LIN {X 0,Y 352.811,Z 516.095,A -85,B 0,C 180,E1 -17555.716,E2 -17555.716} C_VEL
LIN {X 0,Y 351.026,Z 514.823,A -85,B 0,C 180,E1 -17556.899,E2 -17556.899} C_VEL
LIN {X 0,Y 348.295,Z 512.255,A -85,B 0,C 180,E1 -17558.613,E2 -17558.613} C_VEL
LIN {X 0,Y 346.071,Z 510.125,A -85,B 0,C 180,E1 -17559.774,E2 -17559.774} C_VEL
LIN {X 0,Y 342.714,Z 507.631,A -85,B 0,C 180,E1 -17561.14,E2 -17561.14} C_VEL
LIN {X 0,Y 338.592,Z 503.953,A -85,B 0,C 180,E1 -17562.698,E2 -17562.698} C_VEL
LIN {X 0,Y 335.81,Z 501.368,A -85,B 0,C 180,E1 -17563.667,E2 -17563.667} C_VEL
LIN {X 0,Y 331.313,Z 497.271,A -85,B 0,C 180,E1 -17565.061,E2 -17565.061} C_VEL
LIN {X 0,Y 325.512,Z 491.626,A -85,B 0,C 180,E1 -17566.703,E2 -17566.703} C_VEL
LIN {X 0,Y 318.548,Z 484.573,A -85,B 0,C 180,E1 -17568.436,E2 -17568.436} C_VEL
LIN {X 0,Y 312.135,Z 477.632,A -85,B 0,C 180,E1 -17569.889,E2 -17569.889} C_VEL
LIN {X 0,Y 303.985,Z 468.251,A -85,B 0,C 180,E1 -17571.571,E2 -17571.571} C_VEL
LIN {X 0,Y 294.799,Z 456.635,A -85,B 0,C 180,E1 -17573.406,E2 -17573.406} C_VEL
LIN {X 0,Y 287.892,Z 445.985,A -85,B 0,C 180,E1 -17574.797,E2 -17574.797} C_VEL
LIN {X 0,Y 283.079,Z 436.29,A -85,B 0,C 180,E1 -17575.776,E2 -17575.776} C_VEL
LIN {X 0,Y 277.442,Z 424.043,A -85,B 0,C 180,E1 -17576.775,E2 -17576.775} C_VEL
LIN {X 0,Y 277.356,Z 423.437,A -85,B 0,C 180,E1 -17576.824,E2 -17576.824} C_VEL
LIN {X 0,Y 277.267,Z 423.447,A -85,B 0,C 180,E1 -17580.481,E2 -17580.481} C_VEL
LIN {X 0,Y 277.249,Z 423.45,A -85,B 0,C 180,E1 -17583.895,E2 -17583.895} C_VEL
LIN {X 0,Y 277.276,Z 423.448,A -85,B 0,C 180,E1 -17587.467,E2 -17587.467} C_VEL
LIN {X 0,Y 277.204,Z 423.456,A -85,B 0,C 180,E1 -17591.236,E2 -17591.236} C_VEL
LIN {X 0,Y 277.21,Z 423.456,A -85,B 0,C 180,E1 -17595.223,E2 -17595.223} C_VEL
LIN {X 0,Y 277.216,Z 423.454,A -85,B 0,C 180,E1 -17599.512,E2 -17599.512} C_VEL
LIN {X 0,Y 277.258,Z 423.447,A -85,B 0,C 180,E1 -17602.53,E2 -17602.53} C_VEL
LIN {X 0,Y 277.24,Z 423.448,A -85,B 0,C 180,E1 -17606.104,E2 -17606.104} C_VEL
LIN {X 0,Y 277.255,Z 423.448,A -85,B 0,C 180,E1 -17609.539,E2 -17609.539} C_VEL
LIN {X 0,Y 277.352,Z 423.439,A -85,B 0,C 180,E1 -17612.864,E2 -17612.864} C_VEL
LIN {X 0,Y 277.322,Z 423.437,A -85,B 0,C 180,E1 -17616.08,E2 -17616.08} C_VEL
LIN {X 0,Y 277.338,Z 423.436,A -85,B 0,C 180,E1 -17620.767,E2 -17620.767} C_VEL
LIN {X 0,Y 277.421,Z 423.424,A -85,B 0,C 180,E1 -17625.326,E2 -17625.326} C_VEL
LIN {X 0,Y 277.455,Z 423.42,A -85,B 0,C 180,E1 -17629.788,E2 -17629.788} C_VEL
LIN {X 0,Y 277.634,Z 423.404,A -85,B 0,C 180,E1 -17632.729,E2 -17632.729} C_VEL
LIN {X 0,Y 277.815,Z 423.365,A -85,B 0,C 180,E1 -17638.551,E2 -17638.551} C_VEL
LIN {X 0,Y 277.815,Z 423.375,A -85,B 0,C 180,E1 -17641.45,E2 -17641.45} C_VEL
LIN {X 0,Y 277.635,Z 423.4,A -85,B 0,C 180,E1 -17647.272,E2 -17647.272} C_VEL
LIN {X 0,Y 277.456,Z 423.426,A -85,B 0,C 180,E1 -17650.214,E2 -17650.214} C_VEL
LIN {X 0,Y 277.423,Z 423.429,A -85,B 0,C 180,E1 -17654.676,E2 -17654.676} C_VEL
LIN {X 0,Y 277.338,Z 423.437,A -85,B 0,C 180,E1 -17659.235,E2 -17659.235} C_VEL
LIN {X 0,Y 277.289,Z 423.449,A -85,B 0,C 180,E1 -17664.159,E2 -17664.159} C_VEL
LIN {X 0,Y 277.303,Z 423.44,A -85,B 0,C 180,E1 -17666.306,E2 -17666.306} C_VEL
LIN {X 0,Y 276.642,Z 423.527,A -85,B 0,C 180,E1 -17667.519,E2 -17667.519} C_VEL
LIN {X 0,Y 273.724,Z 423.89,A -85,B 0,C 180,E1 -17669.491,E2 -17669.491} C_VEL
LIN {X 0,Y 271.284,Z 424.343,A -85,B 0,C 180,E1 -17671.093,E2 -17671.093} C_VEL
LIN {X 0,Y 270.31,Z 424.816,A -85,B 0,C 180,E1 -17672.334,E2 -17672.334} C_VEL
LIN {X 0,Y 270.27,Z 425.007,A -85,B 0,C 180,E1 -17672.753,E2 -17672.753} C_VEL
LIN {X 0,Y 270.566,Z 427.131,A -85,B 0,C 180,E1 -17676.687,E2 -17676.687} C_VEL
LIN {X 0,Y 270.931,Z 429.384,A -85,B 0,C 180,E1 -17680.43,E2 -17680.43} C_VEL
LIN {X 0,Y 271.232,Z 432.01,A -85,B 0,C 180,E1 -17684.397,E2 -17684.397} C_VEL
LIN {X 0,Y 271.187,Z 434.37,A -85,B 0,C 180,E1 -17687.64,E2 -17687.64} C_VEL
LIN {X 0,Y 270.859,Z 437.105,A -85,B 0,C 180,E1 -17691.117,E2 -17691.117} C_VEL
LIN {X 0,Y 270.245,Z 440.416,A -85,B 0,C 180,E1 -17695.102,E2 -17695.102} C_VEL
LIN {X 0,Y 269.717,Z 443.488,A -85,B 0,C 180,E1 -17698.592,E2 -17698.592} C_VEL
LIN {X 0,Y 269.135,Z 447.13,A -85,B 0,C 180,E1 -17702.656,E2 -17702.656} C_VEL
LIN {X 0,Y 270.056,Z 450.505,A -85,B 0,C 180,E1 -17702.901,E2 -17702.901} C_VEL
LIN {X 0,Y 273.622,Z 464.1,A -85,B 0,C 180,E1 -17704.111,E2 -17704.111} C_VEL
LIN {X 0,Y 275.635,Z 473.958,A -85,B 0,C 180,E1 -17705.134,E2 -17705.134} C_VEL
LIN {X 0,Y 276.955,Z 484.089,A -85,B 0,C 180,E1 -17706.325,E2 -17706.325} C_VEL
LIN {X 0,Y 277.623,Z 492.133,A -85,B 0,C 180,E1 -17707.397,E2 -17707.397} C_VEL
LIN {X 0,Y 277.81,Z 496.843,A -85,B 0,C 180,E1 -17708.091,E2 -17708.091} C_VEL
LIN {X 0,Y 275.735,Z 508.341,A -85,B 0,C 180,E1 -17709.874,E2 -17709.874} C_VEL
LIN {X 0,Y 274.214,Z 516.042,A -85,B 0,C 180,E1 -17711.361,E2 -17711.361} C_VEL
LIN {X 0,Y 272.742,Z 523.682,A -85,B 0,C 180,E1 -17713.149,E2 -17713.149} C_VEL
LIN {X 0,Y 271.421,Z 530.22,A -85,B 0,C 180,E1 -17714.994,E2 -17714.994} C_VEL
LIN {X 0,Y 270.446,Z 534.72,A -85,B 0,C 180,E1 -17716.475,E2 -17716.475} C_VEL
LIN {X 0,Y 269.438,Z 540.214,A -85,B 0,C 180,E1 -17718.719,E2 -17718.719} C_VEL
LIN {X 0,Y 268.752,Z 544.542,A -85,B 0,C 180,E1 -17720.973,E2 -17720.973} C_VEL
LIN {X 0,Y 268.423,Z 546.911,A -85,B 0,C 180,E1 -17722.478,E2 -17722.478} C_VEL
LIN {X 0,Y 268.142,Z 549.611,A -85,B 0,C 180,E1 -17724.867,E2 -17724.867} C_VEL
LIN {X 0,Y 268.168,Z 551.166,A -85,B 0,C 180,E1 -17726.996,E2 -17726.996} C_VEL
LIN {X 0,Y 268.184,Z 551.757,A -85,B 0,C 180,E1 -17728.498,E2 -17728.498} C_VEL
LIN {X 0,Y 268.184,Z 551.757,A -85,B 0,C 180,E1 -17731.502,E2 -17731.502} C_VEL
LIN {X 0,Y 268.169,Z 551.166,A -85,B 0,C 180,E1 -17733.004,E2 -17733.004} C_VEL
LIN {X 0,Y 268.227,Z 548.712,A -85,B 0,C 180,E1 -17736.016,E2 -17736.016} C_VEL
LIN {X 0,Y 268.566,Z 545.76,A -85,B 0,C 180,E1 -17738.275,E2 -17738.275} C_VEL
LIN {X 0,Y 269.201,Z 541.77,A -85,B 0,C 180,E1 -17740.53,E2 -17740.53} C_VEL
LIN {X 0,Y 270.049,Z 536.636,A -85,B 0,C 180,E1 -17742.78,E2 -17742.78} C_VEL
LIN {X 0,Y 271.142,Z 531.374,A -85,B 0,C 180,E1 -17744.638,E2 -17744.638} C_VEL
LIN {X 0,Y 272.187,Z 526.434,A -85,B 0,C 180,E1 -17746.115,E2 -17746.115} C_VEL
LIN {X 0,Y 273.392,Z 520.735,A -85,B 0,C 180,E1 -17747.581,E2 -17747.581} C_VEL
LIN {X 0,Y 274.891,Z 512.177,A -85,B 0,C 180,E1 -17749.412,E2 -17749.412} C_VEL
LIN {X 0,Y 276.5,Z 504,A -85,B 0,C 180,E1 -17750.845,E2 -17750.845} C_VEL
LIN {X 0,Y 277.807,Z 496.842,A -85,B 0,C 180,E1 -17751.909,E2 -17751.909} C_VEL
LIN {X 0,Y 277.292,Z 487.688,A -85,B 0,C 180,E1 -17753.211,E2 -17753.211} C_VEL
LIN {X 0,Y 276.179,Z 477.496,A -85,B 0,C 180,E1 -17754.464,E2 -17754.464} C_VEL
LIN {X 0,Y 274.478,Z 467.955,A -85,B 0,C 180,E1 -17755.501,E2 -17755.501} C_VEL
LIN {X 0,Y 271.905,Z 457.255,A -85,B 0,C 180,E1 -17756.52,E2 -17756.52} C_VEL
LIN {X 0,Y 269.178,Z 447.606,A -85,B 0,C 180,E1 -17757.308,E2 -17757.308} C_VEL
LIN {X 0,Y 269.124,Z 447.099,A -85,B 0,C 180,E1 -17757.39,E2 -17757.39} C_VEL
LIN {X 0,Y 269.717,Z 443.392,A -85,B 0,C 180,E1 -17761.408,E2 -17761.408} C_VEL
LIN {X 0,Y 270.239,Z 440.375,A -85,B 0,C 180,E1 -17764.899,E2 -17764.899} C_VEL
LIN {X 0,Y 270.861,Z 437.075,A -85,B 0,C 180,E1 -17768.884,E2 -17768.884} C_VEL
LIN {X 0,Y 271.208,Z 434.364,A -85,B 0,C 180,E1 -17772.356,E2 -17772.356} C_VEL
LIN {X 0,Y 271.225,Z 432.001,A -85,B 0,C 180,E1 -17775.602,E2 -17775.602} C_VEL
LIN {X 0,Y 270.928,Z 429.377,A -85,B 0,C 180,E1 -17779.57,E2 -17779.57} C_VEL
LIN {X 0,Y 270.543,Z 426.938,A -85,B 0,C 180,E1 -17783.637,E2 -17783.637} C_VEL
LIN {X 0,Y 270.312,Z 425.167,A -85,B 0,C 180,E1 -17786.907,E2 -17786.907} C_VEL
LIN {X 0,Y 270.199,Z 424.332,A -85,B 0,C 180,E1 -17789.129,E2 -17789.129} C_VEL
LIN {X 0,Y 270.262,Z 424.322,A -85,B 0,C 180,E1 -17792.144,E2 -17792.144} C_VEL
LIN {X 0,Y 270.234,Z 424.325,A -85,B 0,C 180,E1 -17795.537,E2 -17795.537} C_VEL
LIN {X 0,Y 270.296,Z 424.316,A -85,B 0,C 180,E1 -17800.243,E2 -17800.243} C_VEL
LIN {X 0,Y 270.392,Z 424.302,A -85,B 0,C 180,E1 -17804.934,E2 -17804.934} C_VEL
LIN {X 0,Y 270.408,Z 424.304,A -85,B 0,C 180,E1 -17809.517,E2 -17809.517} C_VEL
LIN {X 0,Y 270.593,Z 424.276,A -85,B 0,C 180,E1 -17812.538,E2 -17812.538} C_VEL
LIN {X 0,Y 270.781,Z 424.251,A -85,B 0,C 180,E1 -17818.512,E2 -17818.512} C_VEL
LIN {X 0,Y 270.781,Z 424.239,A -85,B 0,C 180,E1 -17821.486,E2 -17821.486} C_VEL
LIN {X 0,Y 270.592,Z 424.28,A -85,B 0,C 180,E1 -17827.461,E2 -17827.461} C_VEL
LIN {X 0,Y 270.406,Z 424.298,A -85,B 0,C 180,E1 -17830.482,E2 -17830.482} C_VEL
LIN {X 0,Y 270.39,Z 424.301,A -85,B 0,C 180,E1 -17835.064,E2 -17835.064} C_VEL
LIN {X 0,Y 270.295,Z 424.311,A -85,B 0,C 180,E1 -17839.755,E2 -17839.755} C_VEL
LIN {X 0,Y 270.268,Z 424.317,A -85,B 0,C 180,E1 -17844.585,E2 -17844.585} C_VEL
LIN {X 0,Y 270.266,Z 424.317,A -85,B 0,C 180,E1 -17847.908,E2 -17847.908} C_VEL
LIN {X 0,Y 270.178,Z 424.33,A -85,B 0,C 180,E1 -17851.348,E2 -17851.348} C_VEL
LIN {X 0,Y 270.209,Z 424.328,A -85,B 0,C 180,E1 -17854.903,E2 -17854.903} C_VEL
LIN {X 0,Y 270.216,Z 424.326,A -85,B 0,C 180,E1 -17858.717,E2 -17858.717} C_VEL
LIN {X 0,Y 270.242,Z 424.324,A -85,B 0,C 180,E1 -17862.543,E2 -17862.543} C_VEL
LIN {X 0,Y 270.183,Z 424.331,A -85,B 0,C 180,E1 -17866.746,E2 -17866.746} C_VEL
LIN {X 0,Y 270.201,Z 424.327,A -85,B 0,C 180,E1 -17871.374,E2 -17871.374} C_VEL
LIN {X 0,Y 270.209,Z 424.327,A -85,B 0,C 180,E1 -17875.097,E2 -17875.097} C_VEL
LIN {X 0,Y 270.195,Z 424.328,A -85,B 0,C 180,E1 -17879.131,E2 -17879.131} C_VEL
LIN {X 0,Y 270.291,Z 424.318,A -85,B 0,C 180,E1 -17882.44,E2 -17882.44} C_VEL
LIN {X 0,Y 271.242,Z 427.063,A -85,B 0,C 180,E1 -17882.645,E2 -17882.645} C_VEL
LIN {X 0,Y 276.988,Z 439.088,A -85,B 0,C 180,E1 -17883.735,E2 -17883.735} C_VEL
LIN {X 0,Y 281.103,Z 447.875,A -85,B 0,C 180,E1 -17884.676,E2 -17884.676} C_VEL
LIN {X 0,Y 286.353,Z 456.735,A -85,B 0,C 180,E1 -17885.846,E2 -17885.846} C_VEL
LIN {X 0,Y 293.982,Z 467.207,A -85,B 0,C 180,E1 -17887.512,E2 -17887.512} C_VEL
LIN {X 0,Y 304.138,Z 479.227,A -85,B 0,C 180,E1 -17889.72,E2 -17889.72} C_VEL
LIN {X 0,Y 312.671,Z 488.513,A -85,B 0,C 180,E1 -17891.659,E2 -17891.659} C_VEL
LIN {X 0,Y 318.131,Z 494.088,A -85,B 0,C 180,E1 -17893.003,E2 -17893.003} C_VEL
LIN {X 0,Y 324.266,Z 500.008,A -85,B 0,C 180,E1 -17894.648,E2 -17894.648} C_VEL
LIN {X 0,Y 330.066,Z 505.438,A -85,B 0,C 180,E1 -17896.455,E2 -17896.455} C_VEL
LIN {X 0,Y 334.025,Z 509.236,A -85,B 0,C 180,E1 -17897.854,E2 -17897.854} C_VEL
LIN {X 0,Y 338.748,Z 513.032,A -85,B 0,C 180,E1 -17899.644,E2 -17899.644} C_VEL
LIN {X 0,Y 341.597,Z 515.35,A -85,B 0,C 180,E1 -17900.944,E2 -17900.944} C_VEL
LIN {X 0,Y 344.939,Z 518.614,A -85,B 0,C 180,E1 -17902.978,E2 -17902.978} C_VEL
LIN {X 0,Y 346.73,Z 519.995,A -85,B 0,C 180,E1 -17904.183,E2 -17904.183} C_VEL
LIN {X 0,Y 348.359,Z 520.945,A -85,B 0,C 180,E1 -17905.371,E2 -17905.371} C_VEL
LIN {X 0,Y 349.735,Z 521.553,A -85,B 0,C 180,E1 -17906.544,E2 -17906.544} C_VEL
LIN {X 0,Y 350.851,Z 521.883,A -85,B 0,C 180,E1 -17907.704,E2 -17907.704} C_VEL
LIN {X 0,Y 351.612,Z 522.025,A -85,B 0,C 180,E1 -17908.855,E2 -17908.855} C_VEL
LIN {X 0,Y 351.859,Z 522.078,A -85,B 0,C 180,E1 -17910,E2 -17910} C_VEL
LIN {X 0,Y 351.482,Z 522.043,A -85,B 0,C 180,E1 -17911.274,E2 -17911.274} C_VEL
LIN {X 0,Y 350.848,Z 521.881,A -85,B 0,C 180,E1 -17912.296,E2 -17912.296} C_VEL
LIN {X 0,Y 349.737,Z 521.547,A -85,B 0,C 180,E1 -17913.456,E2 -17913.456} C_VEL
LIN {X 0,Y 348.369,Z 520.948,A -85,B 0,C 180,E1 -17914.628,E2 -17914.628} C_VEL
LIN {X 0,Y 346.329,Z 519.696,A -85,B 0,C 180,E1 -17916.101,E2 -17916.101} C_VEL
LIN {X 0,Y 342.974,Z 516.792,A -85,B 0,C 180,E1 -17918.247,E2 -17918.247} C_VEL
LIN {X 0,Y 340.695,Z 514.539,A -85,B 0,C 180,E1 -17919.499,E2 -17919.499} C_VEL
LIN {X 0,Y 336.656,Z 511.495,A -85,B 0,C 180,E1 -17921.141,E2 -17921.141} C_VEL
LIN {X 0,Y 333.351,Z 508.557,A -85,B 0,C 180,E1 -17922.398,E2 -17922.398} C_VEL
LIN {X 0,Y 328.67,Z 504.29,A -85,B 0,C 180,E1 -17923.98,E2 -17923.98} C_VEL
LIN {X 0,Y 323.217,Z 499.024,A -85,B 0,C 180,E1 -17925.645,E2 -17925.645} C_VEL
LIN {X 0,Y 316.655,Z 492.581,A -85,B 0,C 180,E1 -17927.379,E2 -17927.379} C_VEL
LIN {X 0,Y 309.448,Z 484.978,A -85,B 0,C 180,E1 -17929.097,E2 -17929.097} C_VEL
LIN {X 0,Y 301.038,Z 475.669,A -85,B 0,C 180,E1 -17930.962,E2 -17930.962} C_VEL
LIN {X 0,Y 291.455,Z 463.927,A -85,B 0,C 180,E1 -17933.036,E2 -17933.036} C_VEL
LIN {X 0,Y 284.677,Z 454.079,A -85,B 0,C 180,E1 -17934.522,E2 -17934.522} C_VEL
LIN {X 0,Y 279.845,Z 445.412,A -85,B 0,C 180,E1 -17935.614,E2 -17935.614} C_VEL
LIN {X 0,Y 273.844,Z 432.334,A -85,B 0,C 180,E1 -17936.893,E2 -17936.893} C_VEL
LIN {X 0,Y 270.474,Z 425.245,A -85,B 0,C 180,E1 -17937.493,E2 -17937.493} C_VEL
LIN {X 0,Y 270.278,Z 424.32,A -85,B 0,C 180,E1 -17937.59,E2 -17937.59} C_VEL
LIN {X 0,Y 270.179,Z 424.332,A -85,B 0,C 180,E1 -17941.348,E2 -17941.348} C_VEL
LIN {X 0,Y 270.209,Z 424.327,A -85,B 0,C 180,E1 -17944.903,E2 -17944.903} C_VEL
LIN {X 0,Y 270.217,Z 424.325,A -85,B 0,C 180,E1 -17948.717,E2 -17948.717} C_VEL
LIN {X 0,Y 270.166,Z 424.333,A -85,B 0,C 180,E1 -17953.25,E2 -17953.25} C_VEL
LIN {X 0,Y 270.168,Z 424.333,A -85,B 0,C 180,E1 -17957.442,E2 -17957.442} C_VEL
LIN {X 0,Y 270.201,Z 424.328,A -85,B 0,C 180,E1 -17961.374,E2 -17961.374} C_VEL
LIN {X 0,Y 270.195,Z 424.33,A -85,B 0,C 180,E1 -17965.095,E2 -17965.095} C_VEL
LIN {X 0,Y 270.194,Z 424.33,A -85,B 0,C 180,E1 -17969.131,E2 -17969.131} C_VEL
LIN {X 0,Y 270.259,Z 424.318,A -85,B 0,C 180,E1 -17972.146,E2 -17972.146} C_VEL
LIN {X 0,Y 270.271,Z 424.316,A -85,B 0,C 180,E1 -17975.52,E2 -17975.52} C_VEL
LIN {X 0,Y 270.295,Z 424.311,A -85,B 0,C 180,E1 -17980.245,E2 -17980.245} C_VEL
LIN {X 0,Y 270.39,Z 424.301,A -85,B 0,C 180,E1 -17984.936,E2 -17984.936} C_VEL
LIN {X 0,Y 270.406,Z 424.298,A -85,B 0,C 180,E1 -17989.518,E2 -17989.518} C_VEL
LIN {X 0,Y 270.592,Z 424.28,A -85,B 0,C 180,E1 -17992.539,E2 -17992.539} C_VEL
LIN {X 0,Y 270.781,Z 424.239,A -85,B 0,C 180,E1 -17998.514,E2 -17998.514} C_VEL
LIN {X 0,Y 270.781,Z 424.251,A -85,B 0,C 180,E1 -18001.488,E2 -18001.488} C_VEL
LIN {X 0,Y 270.593,Z 424.277,A -85,B 0,C 180,E1 -18007.462,E2 -18007.462} C_VEL
LIN {X 0,Y 270.408,Z 424.304,A -85,B 0,C 180,E1 -18010.483,E2 -18010.483} C_VEL
LIN {X 0,Y 270.392,Z 424.303,A -85,B 0,C 180,E1 -18015.066,E2 -18015.066} C_VEL
LIN {X 0,Y 270.296,Z 424.316,A -85,B 0,C 180,E1 -18019.757,E2 -18019.757} C_VEL
LIN {X 0,Y 270.235,Z 424.325,A -85,B 0,C 180,E1 -18024.59,E2 -18024.59} C_VEL
LIN {X 0,Y 270.269,Z 424.321,A -85,B 0,C 180,E1 -18027.91,E2 -18027.91} C_VEL
LIN {X 0,Y 270.188,Z 424.334,A -85,B 0,C 180,E1 -18031.349,E2 -18031.349} C_VEL
LIN {X 0,Y 270.27,Z 425.007,A -85,B 0,C 180,E1 -18032.753,E2 -18032.753} C_VEL
LIN {X 0,Y 269.725,Z 425.745,A -85,B 0,C 180,E1 -18033.99,E2 -18033.99} C_VEL
LIN {X 0,Y 267,Z 427.276,A -85,B 0,C 180,E1 -18036,E2 -18036} C_VEL
LIN {X 0,Y 264.697,Z 428.566,A -85,B 0,C 180,E1 -18037.633,E2 -18037.633} C_VEL
LIN {X 0,Y 263.806,Z 429.451,A -85,B 0,C 180,E1 -18038.899,E2 -18038.899} C_VEL
LIN {X 0,Y 263.789,Z 429.714,A -85,B 0,C 180,E1 -18039.327,E2 -18039.327} C_VEL
LIN {X 0,Y 264.01,Z 431.244,A -85,B 0,C 180,E1 -18041.811,E2 -18041.811} C_VEL
LIN {X 0,Y 264.165,Z 432.745,A -85,B 0,C 180,E1 -18044.085,E2 -18044.085} C_VEL
LIN {X 0,Y 264.192,Z 434.229,A -85,B 0,C 180,E1 -18046.24,E2 -18046.24} C_VEL
LIN {X 0,Y 264.113,Z 435.726,A -85,B 0,C 180,E1 -18048.3,E2 -18048.3} C_VEL
LIN {X 0,Y 263.871,Z 437.477,A -85,B 0,C 180,E1 -18050.57,E2 -18050.57} C_VEL
LIN {X 0,Y 263.321,Z 440.252,A -85,B 0,C 180,E1 -18054.044,E2 -18054.044} C_VEL
LIN {X 0,Y 262.778,Z 443.322,A -85,B 0,C 180,E1 -18057.664,E2 -18057.664} C_VEL
LIN {X 0,Y 262.166,Z 446.678,A -85,B 0,C 180,E1 -18061.563,E2 -18061.563} C_VEL
LIN {X 0,Y 262.146,Z 446.972,A -85,B 0,C 180,E1 -18061.878,E2 -18061.878} C_VEL
LIN {X 0,Y 262.916,Z 450.048,A -85,B 0,C 180,E1 -18062.092,E2 -18062.092} C_VEL
LIN {X 0,Y 266.453,Z 462.719,A -85,B 0,C 180,E1 -18063.265,E2 -18063.265} C_VEL
LIN {X 0,Y 268.77,Z 473.748,A -85,B 0,C 180,E1 -18064.454,E2 -18064.454} C_VEL
LIN {X 0,Y 270.088,Z 483.277,A -85,B 0,C 180,E1 -18065.61,E2 -18065.61} C_VEL
LIN {X 0,Y 270.825,Z 492.155,A -85,B 0,C 180,E1 -18066.831,E2 -18066.831} C_VEL
LIN {X 0,Y 271.007,Z 497.997,A -85,B 0,C 180,E1 -18067.712,E2 -18067.712} C_VEL
LIN {X 0,Y 269.064,Z 508.143,A -85,B 0,C 180,E1 -18069.353,E2 -18069.353} C_VEL
LIN {X 0,Y 267.261,Z 516.833,A -85,B 0,C 180,E1 -18071.099,E2 -18071.099} C_VEL
LIN {X 0,Y 265.949,Z 523.484,A -85,B 0,C 180,E1 -18072.705,E2 -18072.705} C_VEL
LIN {X 0,Y 264.543,Z 530.022,A -85,B 0,C 180,E1 -18074.594,E2 -18074.594} C_VEL
LIN {X 0,Y 263.533,Z 534.522,A -85,B 0,C 180,E1 -18076.113,E2 -18076.113} C_VEL
LIN {X 0,Y 262.443,Z 540.016,A -85,B 0,C 180,E1 -18078.414,E2 -18078.414} C_VEL
LIN {X 0,Y 261.726,Z 544.345,A -85,B 0,C 180,E1 -18080.729,E2 -18080.729} C_VEL
LIN {X 0,Y 261.359,Z 546.713,A -85,B 0,C 180,E1 -18082.273,E2 -18082.273} C_VEL
LIN {X 0,Y 261.043,Z 549.602,A -85,B 0,C 180,E1 -18084.973,E2 -18084.973} C_VEL
LIN {X 0,Y 261.063,Z 550.968,A -85,B 0,C 180,E1 -18086.914,E2 -18086.914} C_VEL
LIN {X 0,Y 261.09,Z 551.56,A -85,B 0,C 180,E1 -18088.458,E2 -18088.458} C_VEL
LIN {X 0,Y 261.127,Z 551.716,A -85,B 0,C 180,E1 -18090,E2 -18090} C_VEL
LIN {X 0,Y 261.09,Z 551.56,A -85,B 0,C 180,E1 -18091.542,E2 -18091.542} C_VEL
LIN {X 0,Y 261.064,Z 550.968,A -85,B 0,C 180,E1 -18093.086,E2 -18093.086} C_VEL
LIN {X 0,Y 261.154,Z 548.515,A -85,B 0,C 180,E1 -18096.179,E2 -18096.179} C_VEL
LIN {X 0,Y 261.53,Z 545.563,A -85,B 0,C 180,E1 -18098.499,E2 -18098.499} C_VEL
LIN {X 0,Y 262.174,Z 541.571,A -85,B 0,C 180,E1 -18100.815,E2 -18100.815} C_VEL
LIN {X 0,Y 263.107,Z 536.438,A -85,B 0,C 180,E1 -18103.123,E2 -18103.123} C_VEL
LIN {X 0,Y 264.262,Z 531.177,A -85,B 0,C 180,E1 -18105.028,E2 -18105.028} C_VEL
LIN {X 0,Y 265.607,Z 524.859,A -85,B 0,C 180,E1 -18106.921,E2 -18106.921} C_VEL
LIN {X 0,Y 266.865,Z 518.908,A -85,B 0,C 180,E1 -18108.422,E2 -18108.422} C_VEL
LIN {X 0,Y 268.178,Z 511.979,A -85,B 0,C 180,E1 -18109.918,E2 -18109.918} C_VEL
LIN {X 0,Y 269.852,Z 503.802,A -85,B 0,C 180,E1 -18111.383,E2 -18111.383} C_VEL
LIN {X 0,Y 270.994,Z 497.997,A -85,B 0,C 180,E1 -18112.289,E2 -18112.289} C_VEL
LIN {X 0,Y 270.467,Z 487.254,A -85,B 0,C 180,E1 -18113.861,E2 -18113.861} C_VEL
LIN {X 0,Y 269.425,Z 477.778,A -85,B 0,C 180,E1 -18115.07,E2 -18115.07} C_VEL
LIN {X 0,Y 267.68,Z 468.336,A -85,B 0,C 180,E1 -18116.15,E2 -18116.15} C_VEL
LIN {X 0,Y 265.263,Z 458.078,A -85,B 0,C 180,E1 -18117.176,E2 -18117.176} C_VEL
LIN {X 0,Y 262.194,Z 447.497,A -85,B 0,C 180,E1 -18118.095,E2 -18118.095} C_VEL
LIN {X 0,Y 262.141,Z 446.947,A -85,B 0,C 180,E1 -18118.154,E2 -18118.154} C_VEL
LIN {X 0,Y 262.613,Z 444.306,A -85,B 0,C 180,E1 -18121.086,E2 -18121.086} C_VEL
LIN {X 0,Y 263.06,Z 441.747,A -85,B 0,C 180,E1 -18124.127,E2 -18124.127} C_VEL
LIN {X 0,Y 263.606,Z 438.712,A -85,B 0,C 180,E1 -18127.82,E2 -18127.82} C_VEL
LIN {X 0,Y 263.906,Z 437.223,A -85,B 0,C 180,E1 -18129.726,E2 -18129.726} C_VEL
LIN {X 0,Y 264.109,Z 435.628,A -85,B 0,C 180,E1 -18131.832,E2 -18131.832} C_VEL
LIN {X 0,Y 264.202,Z 433.988,A -85,B 0,C 180,E1 -18134.091,E2 -18134.091} C_VEL
LIN {X 0,Y 264.125,Z 432.517,A -85,B 0,C 180,E1 -18136.224,E2 -18136.224} C_VEL
LIN {X 0,Y 263.83,Z 429.957,A -85,B 0,C 180,E1 -18140.258,E2 -18140.258} C_VEL
LIN {X 0,Y 263.487,Z 427.756,A -85,B 0,C 180,E1 -18144.068,E2 -18144.068} C_VEL
LIN {X 0,Y 263.215,Z 425.859,A -85,B 0,C 180,E1 -18147.722,E2 -18147.722} C_VEL
LIN {X 0,Y 263.149,Z 425.21,A -85,B 0,C 180,E1 -18149.506,E2 -18149.506} C_VEL
LIN {X 0,Y 263.189,Z 425.201,A -85,B 0,C 180,E1 -18153.001,E2 -18153.001} C_VEL
LIN {X 0,Y 263.151,Z 425.207,A -85,B 0,C 180,E1 -18156.383,E2 -18156.383} C_VEL
LIN {X 0,Y 263.259,Z 425.195,A -85,B 0,C 180,E1 -18159.692,E2 -18159.692} C_VEL
LIN {X 0,Y 263.34,Z 425.181,A -85,B 0,C 180,E1 -18164.521,E2 -18164.521} C_VEL
LIN {X 0,Y 263.35,Z 425.181,A -85,B 0,C 180,E1 -18169.233,E2 -18169.233} C_VEL
LIN {X 0,Y 263.553,Z 425.153,A -85,B 0,C 180,E1 -18172.337,E2 -18172.337} C_VEL
LIN {X 0,Y 263.746,Z 425.127,A -85,B 0,C 180,E1 -18178.472,E2 -18178.472} C_VEL
LIN {X 0,Y 263.746,Z 425.114,A -85,B 0,C 180,E1 -18181.526,E2 -18181.526} C_VEL
LIN {X 0,Y 263.552,Z 425.155,A -85,B 0,C 180,E1 -18187.661,E2 -18187.661} C_VEL
LIN {X 0,Y 263.349,Z 425.178,A -85,B 0,C 180,E1 -18190.766,E2 -18190.766} C_VEL
LIN {X 0,Y 263.338,Z 425.181,A -85,B 0,C 180,E1 -18195.478,E2 -18195.478} C_VEL
LIN {X 0,Y 263.257,Z 425.187,A -85,B 0,C 180,E1 -18200.306,E2 -18200.306} C_VEL
LIN {X 0,Y 263.202,Z 425.197,A -85,B 0,C 180,E1 -18205.291,E2 -18205.291} C_VEL
LIN {X 0,Y 263.174,Z 425.203,A -85,B 0,C 180,E1 -18208.729,E2 -18208.729} C_VEL
LIN {X 0,Y 263.127,Z 425.208,A -85,B 0,C 180,E1 -18212.288,E2 -18212.288} C_VEL
LIN {X 0,Y 263.182,Z 425.199,A -85,B 0,C 180,E1 -18215.978,E2 -18215.978} C_VEL
LIN {X 0,Y 263.155,Z 425.203,A -85,B 0,C 180,E1 -18219.862,E2 -18219.862} C_VEL
LIN {X 0,Y 263.2,Z 425.198,A -85,B 0,C 180,E1 -18221.877,E2 -18221.877} C_VEL
LIN {X 0,Y 263.133,Z 425.207,A -85,B 0,C 180,E1 -18226.147,E2 -18226.147} C_VEL
LIN {X 0,Y 263.111,Z 425.21,A -85,B 0,C 180,E1 -18230.13,E2 -18230.13} C_VEL
LIN {X 0,Y 263.182,Z 425.202,A -85,B 0,C 180,E1 -18234.022,E2 -18234.022} C_VEL
LIN {X 0,Y 263.128,Z 425.208,A -85,B 0,C 180,E1 -18237.712,E2 -18237.712} C_VEL
LIN {X 0,Y 263.22,Z 425.342,A -85,B 0,C 180,E1 -18241.678,E2 -18241.678} C_VEL
LIN {X 0,Y 264.361,Z 428.28,A -85,B 0,C 180,E1 -18241.902,E2 -18241.902} C_VEL
LIN {X 0,Y 270.044,Z 439.972,A -85,B 0,C 180,E1 -18243.044,E2 -18243.044} C_VEL
LIN {X 0,Y 274.293,Z 449.677,A -85,B 0,C 180,E1 -18244.111,E2 -18244.111} C_VEL
LIN {X 0,Y 278.697,Z 457.692,A -85,B 0,C 180,E1 -18245.204,E2 -18245.204} C_VEL
LIN {X 0,Y 285.24,Z 467.472,A -85,B 0,C 180,E1 -18246.783,E2 -18246.783} C_VEL
LIN {X 0,Y 295.013,Z 479.488,A -85,B 0,C 180,E1 -18249.064,E2 -18249.064} C_VEL
LIN {X 0,Y 304.288,Z 489.621,A -85,B 0,C 180,E1 -18251.253,E2 -18251.253} C_VEL
LIN {X 0,Y 312.066,Z 497.676,A -85,B 0,C 180,E1 -18253.158,E2 -18253.158} C_VEL
LIN {X 0,Y 318.593,Z 504.001,A -85,B 0,C 180,E1 -18254.938,E2 -18254.938} C_VEL
LIN {X 0,Y 322.478,Z 507.808,A -85,B 0,C 180,E1 -18256.13,E2 -18256.13} C_VEL
LIN {X 0,Y 326.851,Z 511.751,A -85,B 0,C 180,E1 -18257.583,E2 -18257.583} C_VEL
LIN {X 0,Y 330.568,Z 515.053,A -85,B 0,C 180,E1 -18258.969,E2 -18258.969} C_VEL
LIN {X 0,Y 334.744,Z 518.221,A -85,B 0,C 180,E1 -18260.665,E2 -18260.665} C_VEL
LIN {X 0,Y 336.444,Z 519.881,A -85,B 0,C 180,E1 -18261.592,E2 -18261.592} C_VEL
LIN {X 0,Y 339.503,Z 522.731,A -85,B 0,C 180,E1 -18263.528,E2 -18263.528} C_VEL
LIN {X 0,Y 341.996,Z 524.347,A -85,B 0,C 180,E1 -18265.285,E2 -18265.285} C_VEL
LIN {X 0,Y 343.421,Z 525.041,A -85,B 0,C 180,E1 -18266.48,E2 -18266.48} C_VEL
LIN {X 0,Y 344.647,Z 525.45,A -85,B 0,C 180,E1 -18267.692,E2 -18267.692} C_VEL
LIN {X 0,Y 345.443,Z 525.631,A -85,B 0,C 180,E1 -18268.834,E2 -18268.834} C_VEL
LIN {X 0,Y 345.744,Z 525.684,A -85,B 0,C 180,E1 -18270,E2 -18270} C_VEL
LIN {X 0,Y 345.403,Z 525.651,A -85,B 0,C 180,E1 -18271.166,E2 -18271.166} C_VEL
LIN {X 0,Y 344.618,Z 525.44,A -85,B 0,C 180,E1 -18272.338,E2 -18272.338} C_VEL
LIN {X 0,Y 343.426,Z 525.038,A -85,B 0,C 180,E1 -18273.52,E2 -18273.52} C_VEL
LIN {X 0,Y 342.007,Z 524.353,A -85,B 0,C 180,E1 -18274.715,E2 -18274.715} C_VEL
LIN {X 0,Y 339.501,Z 522.747,A -85,B 0,C 180,E1 -18276.47,E2 -18276.47} C_VEL
LIN {X 0,Y 336.442,Z 519.912,A -85,B 0,C 180,E1 -18278.408,E2 -18278.408} C_VEL
LIN {X 0,Y 333.848,Z 517.577,A -85,B 0,C 180,E1 -18279.695,E2 -18279.695} C_VEL
LIN {X 0,Y 328.714,Z 513.501,A -85,B 0,C 180,E1 -18281.718,E2 -18281.718} C_VEL
LIN {X 0,Y 323.658,Z 508.818,A -85,B 0,C 180,E1 -18283.507,E2 -18283.507} C_VEL
LIN {X 0,Y 318.577,Z 503.994,A -85,B 0,C 180,E1 -18285.074,E2 -18285.074} C_VEL
LIN {X 0,Y 312.054,Z 497.727,A -85,B 0,C 180,E1 -18286.834,E2 -18286.834} C_VEL
LIN {X 0,Y 305.565,Z 491.019,A -85,B 0,C 180,E1 -18288.425,E2 -18288.425} C_VEL
LIN {X 0,Y 297.801,Z 482.616,A -85,B 0,C 180,E1 -18290.271,E2 -18290.271} C_VEL
LIN {X 0,Y 289.661,Z 473.097,A -85,B 0,C 180,E1 -18292.185,E2 -18292.185} C_VEL
LIN {X 0,Y 282.981,Z 464.269,A -85,B 0,C 180,E1 -18293.758,E2 -18293.758} C_VEL
LIN {X 0,Y 276.811,Z 454.544,A -85,B 0,C 180,E1 -18295.249,E2 -18295.249} C_VEL
LIN {X 0,Y 272.212,Z 445.058,A -85,B 0,C 180,E1 -18296.421,E2 -18296.421} C_VEL
LIN {X 0,Y 266.742,Z 432.864,A -85,B 0,C 180,E1 -18297.658,E2 -18297.658} C_VEL
LIN {X 0,Y 263.358,Z 426.118,A -85,B 0,C 180,E1 -18298.282,E2 -18298.282} C_VEL
LIN {X 0,Y 263.191,Z 425.201,A -85,B 0,C 180,E1 -18298.363,E2 -18298.363} C_VEL
LIN {X 0,Y 263.128,Z 425.208,A -85,B 0,C 180,E1 -18302.288,E2 -18302.288} C_VEL
LIN {X 0,Y 263.182,Z 425.202,A -85,B 0,C 180,E1 -18305.978,E2 -18305.978} C_VEL
LIN {X 0,Y 263.11,Z 425.21,A -85,B 0,C 180,E1 -18309.871,E2 -18309.871} C_VEL
LIN {X 0,Y 263.122,Z 425.208,A -85,B 0,C 180,E1 -18313.983,E2 -18313.983} C_VEL
LIN {X 0,Y 263.119,Z 425.208,A -85,B 0,C 180,E1 -18318.406,E2 -18318.406} C_VEL
LIN {X 0,Y 263.175,Z 425.204,A -85,B 0,C 180,E1 -18323.237,E2 -18323.237} C_VEL
LIN {X 0,Y 263.126,Z 425.208,A -85,B 0,C 180,E1 -18327.712,E2 -18327.712} C_VEL
LIN {X 0,Y 263.195,Z 425.198,A -85,B 0,C 180,E1 -18331.783,E2 -18331.783} C_VEL
LIN {X 0,Y 263.22,Z 425.194,A -85,B 0,C 180,E1 -18335.201,E2 -18335.201} C_VEL
LIN {X 0,Y 263.257,Z 425.187,A -85,B 0,C 180,E1 -18339.694,E2 -18339.694} C_VEL
LIN {X 0,Y 263.338,Z 425.181,A -85,B 0,C 180,E1 -18344.522,E2 -18344.522} C_VEL
LIN {X 0,Y 263.349,Z 425.178,A -85,B 0,C 180,E1 -18349.234,E2 -18349.234} C_VEL
LIN {X 0,Y 263.552,Z 425.155,A -85,B 0,C 180,E1 -18352.339,E2 -18352.339} C_VEL
LIN {X 0,Y 263.746,Z 425.114,A -85,B 0,C 180,E1 -18358.474,E2 -18358.474} C_VEL
LIN {X 0,Y 263.746,Z 425.127,A -85,B 0,C 180,E1 -18361.528,E2 -18361.528} C_VEL
LIN {X 0,Y 263.553,Z 425.154,A -85,B 0,C 180,E1 -18367.663,E2 -18367.663} C_VEL
LIN {X 0,Y 263.35,Z 425.182,A -85,B 0,C 180,E1 -18370.767,E2 -18370.767} C_VEL
LIN {X 0,Y 263.34,Z 425.182,A -85,B 0,C 180,E1 -18375.479,E2 -18375.479} C_VEL
LIN {X 0,Y 263.259,Z 425.194,A -85,B 0,C 180,E1 -18380.308,E2 -18380.308} C_VEL
LIN {X 0,Y 263.19,Z 425.202,A -85,B 0,C 180,E1 -18385.294,E2 -18385.294} C_VEL
LIN {X 0,Y 263.177,Z 425.204,A -85,B 0,C 180,E1 -18388.731,E2 -18388.731} C_VEL
LIN {X 0,Y 263.166,Z 425.373,A -85,B 0,C 180,E1 -18391.289,E2 -18391.289} C_VEL
LIN {X 0,Y 263.37,Z 426.831,A -85,B 0,C 180,E1 -18394.187,E2 -18394.187} C_VEL
LIN {X 0,Y 263.636,Z 428.826,A -85,B 0,C 180,E1 -18397.817,E2 -18397.817} C_VEL
LIN {X 0,Y 263.789,Z 429.714,A -85,B 0,C 180,E1 -18399.327,E2 -18399.327} C_VEL
LIN {X 0,Y 263.301,Z 430.568,A -85,B 0,C 180,E1 -18400.589,E2 -18400.589} C_VEL
LIN {X 0,Y 261.844,Z 431.563,A -85,B 0,C 180,E1 -18401.827,E2 -18401.827} C_VEL
LIN {X 0,Y 258.235,Z 433.679,A -85,B 0,C 180,E1 -18404.309,E2 -18404.309} C_VEL
LIN {X 0,Y 257.188,Z 434.686,A -85,B 0,C 180,E1 -18405.601,E2 -18405.601} C_VEL
LIN {X 0,Y 257.095,Z 434.998,A -85,B 0,C 180,E1 -18406.04,E2 -18406.04} C_VEL
LIN {X 0,Y 256.957,Z 437.079,A -85,B 0,C 180,E1 -18408.974,E2 -18408.974} C_VEL
LIN {X 0,Y 256.439,Z 440.088,A -85,B 0,C 180,E1 -18412.921,E2 -18412.921} C_VEL
LIN {X 0,Y 255.828,Z 443.135,A -85,B 0,C 180,E1 -18416.673,E2 -18416.673} C_VEL
LIN {X 0,Y 255.195,Z 446.497,A -85,B 0,C 180,E1 -18420.714,E2 -18420.714} C_VEL
LIN {X 0,Y 255.147,Z 446.777,A -85,B 0,C 180,E1 -18421.032,E2 -18421.032} C_VEL
LIN {X 0,Y 256.057,Z 450.099,A -85,B 0,C 180,E1 -18421.288,E2 -18421.288} C_VEL
LIN {X 0,Y 259.564,Z 462.504,A -85,B 0,C 180,E1 -18422.497,E2 -18422.497} C_VEL
LIN {X 0,Y 261.893,Z 473.536,A -85,B 0,C 180,E1 -18423.733,E2 -18423.733} C_VEL
LIN {X 0,Y 263.265,Z 482.885,A -85,B 0,C 180,E1 -18424.911,E2 -18424.911} C_VEL
LIN {X 0,Y 264.011,Z 492.168,A -85,B 0,C 180,E1 -18426.23,E2 -18426.23} C_VEL
LIN {X 0,Y 264.207,Z 499.06,A -85,B 0,C 180,E1 -18427.313,E2 -18427.313} C_VEL
LIN {X 0,Y 262.398,Z 507.945,A -85,B 0,C 180,E1 -18428.803,E2 -18428.803} C_VEL
LIN {X 0,Y 260.785,Z 515.458,A -85,B 0,C 180,E1 -18430.315,E2 -18430.315} C_VEL
LIN {X 0,Y 259.148,Z 523.382,A -85,B 0,C 180,E1 -18432.264,E2 -18432.264} C_VEL
LIN {X 0,Y 257.673,Z 529.824,A -85,B 0,C 180,E1 -18434.172,E2 -18434.172} C_VEL
LIN {X 0,Y 256.636,Z 534.325,A -85,B 0,C 180,E1 -18435.732,E2 -18435.732} C_VEL
LIN {X 0,Y 255.461,Z 539.818,A -85,B 0,C 180,E1 -18438.093,E2 -18438.093} C_VEL
LIN {X 0,Y 254.683,Z 544.147,A -85,B 0,C 180,E1 -18440.47,E2 -18440.47} C_VEL
LIN {X 0,Y 254.318,Z 546.516,A -85,B 0,C 180,E1 -18442.058,E2 -18442.058} C_VEL
LIN {X 0,Y 253.949,Z 549.585,A -85,B 0,C 180,E1 -18445.073,E2 -18445.073} C_VEL
LIN {X 0,Y 253.962,Z 550.771,A -85,B 0,C 180,E1 -18446.827,E2 -18446.827} C_VEL
LIN {X 0,Y 253.997,Z 551.363,A -85,B 0,C 180,E1 -18448.414,E2 -18448.414} C_VEL
LIN {X 0,Y 254.054,Z 551.519,A -85,B 0,C 180,E1 -18450,E2 -18450} C_VEL
LIN {X 0,Y 253.998,Z 551.363,A -85,B 0,C 180,E1 -18451.586,E2 -18451.586} C_VEL
LIN {X 0,Y 253.964,Z 550.771,A -85,B 0,C 180,E1 -18453.173,E2 -18453.173} C_VEL
LIN {X 0,Y 254.067,Z 548.317,A -85,B 0,C 180,E1 -18456.353,E2 -18456.353} C_VEL
LIN {X 0,Y 254.487,Z 545.365,A -85,B 0,C 180,E1 -18458.736,E2 -18458.736} C_VEL
LIN {X 0,Y 255.16,Z 541.373,A -85,B 0,C 180,E1 -18461.116,E2 -18461.116} C_VEL
LIN {X 0,Y 256.182,Z 536.241,A -85,B 0,C 180,E1 -18463.484,E2 -18463.484} C_VEL
LIN {X 0,Y 257.396,Z 530.979,A -85,B 0,C 180,E1 -18465.439,E2 -18465.439} C_VEL
LIN {X 0,Y 258.81,Z 524.662,A -85,B 0,C 180,E1 -18467.379,E2 -18467.379} C_VEL
LIN {X 0,Y 260.09,Z 518.561,A -85,B 0,C 180,E1 -18468.957,E2 -18468.957} C_VEL
LIN {X 0,Y 261.506,Z 511.782,A -85,B 0,C 180,E1 -18470.449,E2 -18470.449} C_VEL
LIN {X 0,Y 263.251,Z 503.605,A -85,B 0,C 180,E1 -18471.947,E2 -18471.947} C_VEL
LIN {X 0,Y 264.27,Z 497.794,A -85,B 0,C 180,E1 -18472.888,E2 -18472.888} C_VEL
LIN {X 0,Y 263.65,Z 487.046,A -85,B 0,C 180,E1 -18474.518,E2 -18474.518} C_VEL
LIN {X 0,Y 262.659,Z 478.044,A -85,B 0,C 180,E1 -18475.712,E2 -18475.712} C_VEL
LIN {X 0,Y 260.7,Z 467.455,A -85,B 0,C 180,E1 -18476.961,E2 -18476.961} C_VEL
LIN {X 0,Y 258.141,Z 457.132,A -85,B 0,C 180,E1 -18478.036,E2 -18478.036} C_VEL
LIN {X 0,Y 255.241,Z 447.534,A -85,B 0,C 180,E1 -18478.92,E2 -18478.92} C_VEL
LIN {X 0,Y 255.15,Z 446.793,A -85,B 0,C 180,E1 -18478.968,E2 -18478.968} C_VEL
LIN {X 0,Y 255.581,Z 444.563,A -85,B 0,C 180,E1 -18481.52,E2 -18481.52} C_VEL
LIN {X 0,Y 256.128,Z 441.585,A -85,B 0,C 180,E1 -18485.185,E2 -18485.185} C_VEL
LIN {X 0,Y 256.736,Z 438.573,A -85,B 0,C 180,E1 -18489.02,E2 -18489.02} C_VEL
LIN {X 0,Y 257.074,Z 436.061,A -85,B 0,C 180,E1 -18492.426,E2 -18492.426} C_VEL
LIN {X 0,Y 257.122,Z 434.078,A -85,B 0,C 180,E1 -18495.288,E2 -18495.288} C_VEL
LIN {X 0,Y 256.873,Z 431.747,A -85,B 0,C 180,E1 -18498.955,E2 -18498.955} C_VEL
LIN {X 0,Y 256.535,Z 429.428,A -85,B 0,C 180,E1 -18502.935,E2 -18502.935} C_VEL
LIN {X 0,Y 256.262,Z 427.435,A -85,B 0,C 180,E1 -18506.735,E2 -18506.735} C_VEL
LIN {X 0,Y 256.16,Z 426.543,A -85,B 0,C 180,E1 -18508.581,E2 -18508.581} C_VEL
LIN {X 0,Y 256.136,Z 426.082,A -85,B 0,C 180,E1 -18511.404,E2 -18511.404} C_VEL
LIN {X 0,Y 256.14,Z 426.082,A -85,B 0,C 180,E1 -18515.695,E2 -18515.695} C_VEL
LIN {X 0,Y 256.159,Z 426.077,A -85,B 0,C 180,E1 -18519.103,E2 -18519.103} C_VEL
LIN {X 0,Y 256.276,Z 426.063,A -85,B 0,C 180,E1 -18524.083,E2 -18524.083} C_VEL
LIN {X 0,Y 256.289,Z 426.061,A -85,B 0,C 180,E1 -18527.327,E2 -18527.327} C_VEL
LIN {X 0,Y 256.51,Z 426.031,A -85,B 0,C 180,E1 -18532.125,E2 -18532.125} C_VEL
LIN {X 0,Y 256.494,Z 426.034,A -85,B 0,C 180,E1 -18536.858,E2 -18536.858} C_VEL
LIN {X 0,Y 256.759,Z 425.99,A -85,B 0,C 180,E1 -18539.999,E2 -18539.999} C_VEL
LIN {X 0,Y 256.493,Z 426.02,A -85,B 0,C 180,E1 -18543.141,E2 -18543.141} C_VEL
LIN {X 0,Y 256.509,Z 426.031,A -85,B 0,C 180,E1 -18547.873,E2 -18547.873} C_VEL
LIN {X 0,Y 256.287,Z 426.06,A -85,B 0,C 180,E1 -18552.672,E2 -18552.672} C_VEL
LIN {X 0,Y 256.272,Z 426.06,A -85,B 0,C 180,E1 -18556.298,E2 -18556.298} C_VEL
LIN {X 0,Y 256.151,Z 426.076,A -85,B 0,C 180,E1 -18561.119,E2 -18561.119} C_VEL
LIN {X 0,Y 256.182,Z 426.071,A -85,B 0,C 180,E1 -18565.138,E2 -18565.138} C_VEL
LIN {X 0,Y 256.108,Z 426.082,A -85,B 0,C 180,E1 -18569.599,E2 -18569.599} C_VEL
LIN {X 0,Y 256.079,Z 426.087,A -85,B 0,C 180,E1 -18573.29,E2 -18573.29} C_VEL
LIN {X 0,Y 256.134,Z 426.079,A -85,B 0,C 180,E1 -18577.278,E2 -18577.278} C_VEL
LIN {X 0,Y 256.125,Z 426.081,A -85,B 0,C 180,E1 -18581.188,E2 -18581.188} C_VEL
LIN {X 0,Y 256.067,Z 426.087,A -85,B 0,C 180,E1 -18585.527,E2 -18585.527} C_VEL
LIN {X 0,Y 256.056,Z 426.09,A -85,B 0,C 180,E1 -18588.798,E2 -18588.798} C_VEL
LIN {X 0,Y 256.14,Z 426.08,A -85,B 0,C 180,E1 -18592.87,E2 -18592.87} C_VEL
LIN {X 0,Y 256.08,Z 426.088,A -85,B 0,C 180,E1 -18596.71,E2 -18596.71} C_VEL
LIN {X 0,Y 256.098,Z 426.085,A -85,B 0,C 180,E1 -18600.823,E2 -18600.823} C_VEL
LIN {X 0,Y 257.039,Z 428.793,A -85,B 0,C 180,E1 -18601.037,E2 -18601.037} C_VEL
LIN {X 0,Y 261.108,Z 436.611,A -85,B 0,C 180,E1 -18601.853,E2 -18601.853} C_VEL
LIN {X 0,Y 266.582,Z 449.278,A -85,B 0,C 180,E1 -18603.258,E2 -18603.258} C_VEL
LIN {X 0,Y 271.37,Z 459.086,A -85,B 0,C 180,E1 -18604.597,E2 -18604.597} C_VEL
LIN {X 0,Y 278.071,Z 469.65,A -85,B 0,C 180,E1 -18606.372,E2 -18606.372} C_VEL
LIN {X 0,Y 286.851,Z 480.803,A -85,B 0,C 180,E1 -18608.592,E2 -18608.592} C_VEL
LIN {X 0,Y 295.72,Z 490.579,A -85,B 0,C 180,E1 -18610.81,E2 -18610.81} C_VEL
LIN {X 0,Y 304.813,Z 499.855,A -85,B 0,C 180,E1 -18613.105,E2 -18613.105} C_VEL
LIN {X 0,Y 311.27,Z 506.151,A -85,B 0,C 180,E1 -18614.842,E2 -18614.842} C_VEL
LIN {X 0,Y 316.658,Z 511.333,A -85,B 0,C 180,E1 -18616.489,E2 -18616.489} C_VEL
LIN {X 0,Y 321.217,Z 515.492,A -85,B 0,C 180,E1 -18618.004,E2 -18618.004} C_VEL
LIN {X 0,Y 324.914,Z 518.664,A -85,B 0,C 180,E1 -18619.406,E2 -18619.406} C_VEL
LIN {X 0,Y 327.737,Z 520.866,A -85,B 0,C 180,E1 -18620.543,E2 -18620.543} C_VEL
LIN {X 0,Y 330.65,Z 523.554,A -85,B 0,C 180,E1 -18622.059,E2 -18622.059} C_VEL
LIN {X 0,Y 333.578,Z 526.102,A -85,B 0,C 180,E1 -18623.953,E2 -18623.953} C_VEL
LIN {X 0,Y 335.325,Z 527.219,A -85,B 0,C 180,E1 -18625.191,E2 -18625.191} C_VEL
LIN {X 0,Y 337.727,Z 528.392,A -85,B 0,C 180,E1 -18627.252,E2 -18627.252} C_VEL
LIN {X 0,Y 339.019,Z 528.741,A -85,B 0,C 180,E1 -18628.812,E2 -18628.812} C_VEL
LIN {X 0,Y 339.373,Z 528.807,A -85,B 0,C 180,E1 -18630,E2 -18630} C_VEL
LIN {X 0,Y 338.991,Z 528.751,A -85,B 0,C 180,E1 -18631.188,E2 -18631.188} C_VEL
LIN {X 0,Y 337.731,Z 528.383,A -85,B 0,C 180,E1 -18632.761,E2 -18632.761} C_VEL
LIN {X 0,Y 335.333,Z 527.23,A -85,B 0,C 180,E1 -18634.809,E2 -18634.809} C_VEL
LIN {X 0,Y 332.591,Z 525.329,A -85,B 0,C 180,E1 -18636.713,E2 -18636.713} C_VEL
LIN {X 0,Y 329.512,Z 522.445,A -85,B 0,C 180,E1 -18638.586,E2 -18638.586} C_VEL
LIN {X 0,Y 326.579,Z 519.99,A -85,B 0,C 180,E1 -18639.913,E2 -18639.913} C_VEL
LIN {X 0,Y 322.664,Z 516.811,A -85,B 0,C 180,E1 -18641.439,E2 -18641.439} C_VEL
LIN {X 0,Y 317.644,Z 512.209,A -85,B 0,C 180,E1 -18643.219,E2 -18643.219} C_VEL
LIN {X 0,Y 311.266,Z 506.155,A -85,B 0,C 180,E1 -18645.155,E2 -18645.155} C_VEL
LIN {X 0,Y 303.517,Z 498.561,A -85,B 0,C 180,E1 -18647.227,E2 -18647.227} C_VEL
LIN {X 0,Y 293.214,Z 487.972,A -85,B 0,C 180,E1 -18649.82,E2 -18649.82} C_VEL
LIN {X 0,Y 283.32,Z 476.512,A -85,B 0,C 180,E1 -18652.298,E2 -18652.298} C_VEL
LIN {X 0,Y 276.791,Z 467.73,A -85,B 0,C 180,E1 -18653.969,E2 -18653.969} C_VEL
LIN {X 0,Y 270.746,Z 457.937,A -85,B 0,C 180,E1 -18655.576,E2 -18655.576} C_VEL
LIN {X 0,Y 266.301,Z 448.474,A -85,B 0,C 180,E1 -18656.832,E2 -18656.832} C_VEL
LIN {X 0,Y 260.461,Z 435.184,A -85,B 0,C 180,E1 -18658.294,E2 -18658.294} C_VEL
LIN {X 0,Y 256.359,Z 427.325,A -85,B 0,C 180,E1 -18659.096,E2 -18659.096} C_VEL
LIN {X 0,Y 256.1,Z 426.085,A -85,B 0,C 180,E1 -18659.177,E2 -18659.177} C_VEL
LIN {X 0,Y 256.08,Z 426.088,A -85,B 0,C 180,E1 -18663.29,E2 -18663.29} C_VEL
LIN {X 0,Y 256.123,Z 426.083,A -85,B 0,C 180,E1 -18667.275,E2 -18667.275} C_VEL
LIN {X 0,Y 256.052,Z 426.091,A -85,B 0,C 180,E1 -18671.203,E2 -18671.203} C_VEL
LIN {X 0,Y 256.056,Z 426.091,A -85,B 0,C 180,E1 -18675.529,E2 -18675.529} C_VEL
LIN {X 0,Y 256.049,Z 426.091,A -85,B 0,C 180,E1 -18678.797,E2 -18678.797} C_VEL
LIN {X 0,Y 256.123,Z 426.081,A -85,B 0,C 180,E1 -18682.867,E2 -18682.867} C_VEL
LIN {X 0,Y 256.062,Z 426.089,A -85,B 0,C 180,E1 -18686.707,E2 -18686.707} C_VEL
LIN {X 0,Y 256.108,Z 426.082,A -85,B 0,C 180,E1 -18690.401,E2 -18690.401} C_VEL
LIN {X 0,Y 256.182,Z 426.071,A -85,B 0,C 180,E1 -18694.862,E2 -18694.862} C_VEL
LIN {X 0,Y 256.161,Z 426.073,A -85,B 0,C 180,E1 -18699.105,E2 -18699.105} C_VEL
LIN {X 0,Y 256.288,Z 426.058,A -85,B 0,C 180,E1 -18704.085,E2 -18704.085} C_VEL
LIN {X 0,Y 256.287,Z 426.06,A -85,B 0,C 180,E1 -18707.328,E2 -18707.328} C_VEL
LIN {X 0,Y 256.509,Z 426.031,A -85,B 0,C 180,E1 -18712.127,E2 -18712.127} C_VEL
LIN {X 0,Y 256.493,Z 426.02,A -85,B 0,C 180,E1 -18716.859,E2 -18716.859} C_VEL
LIN {X 0,Y 256.759,Z 425.99,A -85,B 0,C 180,E1 -18720.001,E2 -18720.001} C_VEL
LIN {X 0,Y 256.494,Z 426.034,A -85,B 0,C 180,E1 -18723.142,E2 -18723.142} C_VEL
LIN {X 0,Y 256.51,Z 426.033,A -85,B 0,C 180,E1 -18727.875,E2 -18727.875} C_VEL
LIN {X 0,Y 256.289,Z 426.062,A -85,B 0,C 180,E1 -18732.673,E2 -18732.673} C_VEL
LIN {X 0,Y 256.257,Z 426.067,A -85,B 0,C 180,E1 -18736.286,E2 -18736.286} C_VEL
LIN {X 0,Y 256.159,Z 426.076,A -85,B 0,C 180,E1 -18740.897,E2 -18740.897} C_VEL
LIN {X 0,Y 256.168,Z 426.077,A -85,B 0,C 180,E1 -18745.131,E2 -18745.131} C_VEL
LIN {X 0,Y 256.112,Z 426.084,A -85,B 0,C 180,E1 -18749.601,E2 -18749.601} C_VEL
LIN {X 0,Y 256.185,Z 426.699,A -85,B 0,C 180,E1 -18751.744,E2 -18751.744} C_VEL
LIN {X 0,Y 256.401,Z 428.404,A -85,B 0,C 180,E1 -18755.144,E2 -18755.144} C_VEL
LIN {X 0,Y 256.741,Z 430.724,A -85,B 0,C 180,E1 -18759.324,E2 -18759.324} C_VEL
LIN {X 0,Y 257.045,Z 433.048,A -85,B 0,C 180,E1 -18763.122,E2 -18763.122} C_VEL
LIN {X 0,Y 257.095,Z 434.998,A -85,B 0,C 180,E1 -18766.04,E2 -18766.04} C_VEL
LIN {X 0,Y 256.376,Z 435.981,A -85,B 0,C 180,E1 -18767.327,E2 -18767.327} C_VEL
LIN {X 0,Y 253.36,Z 437.819,A -85,B 0,C 180,E1 -18769.408,E2 -18769.408} C_VEL
LIN {X 0,Y 250.729,Z 439.343,A -85,B 0,C 180,E1 -18771.099,E2 -18771.099} C_VEL
LIN {X 0,Y 249.491,Z 440.45,A -85,B 0,C 180,E1 -18772.418,E2 -18772.418} C_VEL
LIN {X 0,Y 249.333,Z 440.804,A -85,B 0,C 180,E1 -18772.867,E2 -18772.867} C_VEL
LIN {X 0,Y 248.933,Z 442.947,A -85,B 0,C 180,E1 -18775.623,E2 -18775.623} C_VEL
LIN {X 0,Y 248.234,Z 446.523,A -85,B 0,C 180,E1 -18780.06,E2 -18780.06} C_VEL
LIN {X 0,Y 248.234,Z 446.808,A -85,B 0,C 180,E1 -18780.16,E2 -18780.16} C_VEL
LIN {X 0,Y 249.898,Z 452.62,A -85,B 0,C 180,E1 -18780.673,E2 -18780.673} C_VEL
LIN {X 0,Y 252.948,Z 463.456,A -85,B 0,C 180,E1 -18781.815,E2 -18781.815} C_VEL
LIN {X 0,Y 255.102,Z 473.756,A -85,B 0,C 180,E1 -18783.025,E2 -18783.025} C_VEL
LIN {X 0,Y 256.579,Z 483.3,A -85,B 0,C 180,E1 -18784.292,E2 -18784.292} C_VEL
LIN {X 0,Y 257.246,Z 492.183,A -85,B 0,C 180,E1 -18785.599,E2 -18785.599} C_VEL
LIN {X 0,Y 257.411,Z 500.005,A -85,B 0,C 180,E1 -18786.892,E2 -18786.892} C_VEL
LIN {X 0,Y 255.762,Z 507.747,A -85,B 0,C 180,E1 -18788.226,E2 -18788.226} C_VEL
LIN {X 0,Y 253.709,Z 516.884,A -85,B 0,C 180,E1 -18790.164,E2 -18790.164} C_VEL
LIN {X 0,Y 252.041,Z 524.465,A -85,B 0,C 180,E1 -18792.138,E2 -18792.138} C_VEL
LIN {X 0,Y 250.538,Z 530.782,A -85,B 0,C 180,E1 -18794.128,E2 -18794.128} C_VEL
LIN {X 0,Y 249.243,Z 536.042,A -85,B 0,C 180,E1 -18796.133,E2 -18796.133} C_VEL
LIN {X 0,Y 248.165,Z 541.175,A -85,B 0,C 180,E1 -18798.566,E2 -18798.566} C_VEL
LIN {X 0,Y 247.459,Z 545.167,A -85,B 0,C 180,E1 -18801.014,E2 -18801.014} C_VEL
LIN {X 0,Y 247.012,Z 548.12,A -85,B 0,C 180,E1 -18803.465,E2 -18803.465} C_VEL
LIN {X 0,Y 246.865,Z 550.573,A -85,B 0,C 180,E1 -18806.736,E2 -18806.736} C_VEL
LIN {X 0,Y 246.907,Z 551.166,A -85,B 0,C 180,E1 -18808.369,E2 -18808.369} C_VEL
LIN {X 0,Y 246.983,Z 551.323,A -85,B 0,C 180,E1 -18810,E2 -18810} C_VEL
LIN {X 0,Y 246.907,Z 551.166,A -85,B 0,C 180,E1 -18811.631,E2 -18811.631} C_VEL
LIN {X 0,Y 246.866,Z 550.573,A -85,B 0,C 180,E1 -18813.264,E2 -18813.264} C_VEL
LIN {X 0,Y 247.012,Z 548.12,A -85,B 0,C 180,E1 -18816.535,E2 -18816.535} C_VEL
LIN {X 0,Y 247.459,Z 545.167,A -85,B 0,C 180,E1 -18818.986,E2 -18818.986} C_VEL
LIN {X 0,Y 248.165,Z 541.175,A -85,B 0,C 180,E1 -18821.434,E2 -18821.434} C_VEL
LIN {X 0,Y 249.243,Z 536.042,A -85,B 0,C 180,E1 -18823.867,E2 -18823.867} C_VEL
LIN {X 0,Y 250.541,Z 530.782,A -85,B 0,C 180,E1 -18825.872,E2 -18825.872} C_VEL
LIN {X 0,Y 252.037,Z 524.465,A -85,B 0,C 180,E1 -18827.862,E2 -18827.862} C_VEL
LIN {X 0,Y 253.676,Z 516.883,A -85,B 0,C 180,E1 -18829.839,E2 -18829.839} C_VEL
LIN {X 0,Y 255.717,Z 507.746,A -85,B 0,C 180,E1 -18831.778,E2 -18831.778} C_VEL
LIN {X 0,Y 257.501,Z 498.858,A -85,B 0,C 180,E1 -18833.312,E2 -18833.312} C_VEL
LIN {X 0,Y 257.082,Z 489.158,A -85,B 0,C 180,E1 -18834.881,E2 -18834.881} C_VEL
LIN {X 0,Y 255.884,Z 478.337,A -85,B 0,C 180,E1 -18836.391,E2 -18836.391} C_VEL
LIN {X 0,Y 253.966,Z 467.886,A -85,B 0,C 180,E1 -18837.681,E2 -18837.681} C_VEL
LIN {X 0,Y 251.407,Z 457.635,A -85,B 0,C 180,E1 -18838.809,E2 -18838.809} C_VEL
LIN {X 0,Y 248.287,Z 447.338,A -85,B 0,C 180,E1 -18839.81,E2 -18839.81} C_VEL
LIN {X 0,Y 248.221,Z 446.601,A -85,B 0,C 180,E1 -18839.873,E2 -18839.873} C_VEL
LIN {X 0,Y 248.621,Z 444.404,A -85,B 0,C 180,E1 -18842.485,E2 -18842.485} C_VEL
LIN {X 0,Y 249.214,Z 441.421,A -85,B 0,C 180,E1 -18846.313,E2 -18846.313} C_VEL
LIN {X 0,Y 249.856,Z 438.412,A -85,B 0,C 180,E1 -18850.311,E2 -18850.311} C_VEL
LIN {X 0,Y 250.068,Z 436.48,A -85,B 0,C 180,E1 -18853.053,E2 -18853.053} C_VEL
LIN {X 0,Y 250.092,Z 434.932,A -85,B 0,C 180,E1 -18855.368,E2 -18855.368} C_VEL
LIN {X 0,Y 249.825,Z 432.443,A -85,B 0,C 180,E1 -18859.423,E2 -18859.423} C_VEL
LIN {X 0,Y 249.436,Z 430.046,A -85,B 0,C 180,E1 -18863.722,E2 -18863.722} C_VEL
LIN {X 0,Y 249.19,Z 428.017,A -85,B 0,C 180,E1 -18867.788,E2 -18867.788} C_VEL
LIN {X 0,Y 249.084,Z 427.243,A -85,B 0,C 180,E1 -18869.477,E2 -18869.477} C_VEL
LIN {X 0,Y 249.095,Z 426.959,A -85,B 0,C 180,E1 -18871.337,E2 -18871.337} C_VEL
LIN {X 0,Y 249.132,Z 426.952,A -85,B 0,C 180,E1 -18874.965,E2 -18874.965} C_VEL
LIN {X 0,Y 249.104,Z 426.957,A -85,B 0,C 180,E1 -18880.21,E2 -18880.21} C_VEL
LIN {X 0,Y 249.22,Z 426.943,A -85,B 0,C 180,E1 -18883.619,E2 -18883.619} C_VEL
LIN {X 0,Y 249.24,Z 426.937,A -85,B 0,C 180,E1 -18888.615,E2 -18888.615} C_VEL
LIN {X 0,Y 249.45,Z 426.912,A -85,B 0,C 180,E1 -18891.901,E2 -18891.901} C_VEL
LIN {X 0,Y 249.292,Z 426.932,A -85,B 0,C 180,E1 -18895.148,E2 -18895.148} C_VEL
LIN {X 0,Y 249.671,Z 426.88,A -85,B 0,C 180,E1 -18898.386,E2 -18898.386} C_VEL
LIN {X 0,Y 249.67,Z 426.864,A -85,B 0,C 180,E1 -18901.612,E2 -18901.612} C_VEL
LIN {X 0,Y 249.435,Z 426.911,A -85,B 0,C 180,E1 -18906.71,E2 -18906.71} C_VEL
LIN {X 0,Y 249.338,Z 426.923,A -85,B 0,C 180,E1 -18909.736,E2 -18909.736} C_VEL
LIN {X 0,Y 249.195,Z 426.94,A -85,B 0,C 180,E1 -18914.703,E2 -18914.703} C_VEL
LIN {X 0,Y 249.133,Z 426.95,A -85,B 0,C 180,E1 -18918.077,E2 -18918.077} C_VEL
LIN {X 0,Y 249.081,Z 426.958,A -85,B 0,C 180,E1 -18921.518,E2 -18921.518} C_VEL
LIN {X 0,Y 249.125,Z 426.951,A -85,B 0,C 180,E1 -18925.482,E2 -18925.482} C_VEL
LIN {X 0,Y 249.077,Z 426.96,A -85,B 0,C 180,E1 -18928.993,E2 -18928.993} C_VEL
LIN {X 0,Y 249.03,Z 426.964,A -85,B 0,C 180,E1 -18932.425,E2 -18932.425} C_VEL
LIN {X 0,Y 249.068,Z 426.958,A -85,B 0,C 180,E1 -18936.338,E2 -18936.338} C_VEL
LIN {X 0,Y 249.078,Z 426.959,A -85,B 0,C 180,E1 -18940.463,E2 -18940.463} C_VEL
LIN {X 0,Y 249.068,Z 426.96,A -85,B 0,C 180,E1 -18942.808,E2 -18942.808} C_VEL
LIN {X 0,Y 249.019,Z 426.965,A -85,B 0,C 180,E1 -18947.365,E2 -18947.365} C_VEL
LIN {X 0,Y 249.034,Z 426.964,A -85,B 0,C 180,E1 -18951.622,E2 -18951.622} C_VEL
LIN {X 0,Y 249.056,Z 426.961,A -85,B 0,C 180,E1 -18955.642,E2 -18955.642} C_VEL
LIN {X 0,Y 249.038,Z 426.985,A -85,B 0,C 180,E1 -18959.943,E2 -18959.943} C_VEL
LIN {X 0,Y 250.048,Z 429.781,A -85,B 0,C 180,E1 -18960.179,E2 -18960.179} C_VEL
LIN {X 0,Y 255.652,Z 440.679,A -85,B 0,C 180,E1 -18961.408,E2 -18961.408} C_VEL
LIN {X 0,Y 259.988,Z 451.008,A -85,B 0,C 180,E1 -18962.643,E2 -18962.643} C_VEL
LIN {X 0,Y 263.743,Z 459.513,A -85,B 0,C 180,E1 -18963.826,E2 -18963.826} C_VEL
LIN {X 0,Y 269.209,Z 469.147,A -85,B 0,C 180,E1 -18965.453,E2 -18965.453} C_VEL
LIN {X 0,Y 276.037,Z 478.706,A -85,B 0,C 180,E1 -18967.357,E2 -18967.357} C_VEL
LIN {X 0,Y 285.22,Z 489.5,A -85,B 0,C 180,E1 -18969.821,E2 -18969.821} C_VEL
LIN {X 0,Y 294.923,Z 499.544,A -85,B 0,C 180,E1 -18972.398,E2 -18972.398} C_VEL
LIN {X 0,Y 302.656,Z 506.947,A -85,B 0,C 180,E1 -18974.506,E2 -18974.506} C_VEL
LIN {X 0,Y 308.908,Z 512.829,A -85,B 0,C 180,E1 -18976.34,E2 -18976.34} C_VEL
LIN {X 0,Y 315.234,Z 518.559,A -85,B 0,C 180,E1 -18978.425,E2 -18978.425} C_VEL
LIN {X 0,Y 320.649,Z 523.023,A -85,B 0,C 180,E1 -18980.504,E2 -18980.504} C_VEL
LIN {X 0,Y 323.486,Z 525.517,A -85,B 0,C 180,E1 -18981.882,E2 -18981.882} C_VEL
LIN {X 0,Y 326.568,Z 528.245,A -85,B 0,C 180,E1 -18983.823,E2 -18983.823} C_VEL
LIN {X 0,Y 328.384,Z 529.547,A -85,B 0,C 180,E1 -18985.089,E2 -18985.089} C_VEL
LIN {X 0,Y 330.765,Z 530.83,A -85,B 0,C 180,E1 -18986.999,E2 -18986.999} C_VEL
LIN {X 0,Y 332.363,Z 531.336,A -85,B 0,C 180,E1 -18988.788,E2 -18988.788} C_VEL
LIN {X 0,Y 332.762,Z 531.416,A -85,B 0,C 180,E1 -18990,E2 -18990} C_VEL
LIN {X 0,Y 332.342,Z 531.341,A -85,B 0,C 180,E1 -18991.212,E2 -18991.212} C_VEL
LIN {X 0,Y 330.765,Z 530.829,A -85,B 0,C 180,E1 -18993.001,E2 -18993.001} C_VEL
LIN {X 0,Y 328.407,Z 529.549,A -85,B 0,C 180,E1 -18994.91,E2 -18994.91} C_VEL
LIN {X 0,Y 325.59,Z 527.446,A -85,B 0,C 180,E1 -18996.825,E2 -18996.825} C_VEL
LIN {X 0,Y 323.478,Z 525.533,A -85,B 0,C 180,E1 -18998.118,E2 -18998.118} C_VEL
LIN {X 0,Y 320.63,Z 523.04,A -85,B 0,C 180,E1 -18999.475,E2 -18999.475} C_VEL
LIN {X 0,Y 315.234,Z 518.537,A -85,B 0,C 180,E1 -19001.575,E2 -19001.575} C_VEL
LIN {X 0,Y 308.928,Z 512.833,A -85,B 0,C 180,E1 -19003.658,E2 -19003.658} C_VEL
LIN {X 0,Y 302.665,Z 506.916,A -85,B 0,C 180,E1 -19005.5,E2 -19005.5} C_VEL
LIN {X 0,Y 293.764,Z 498.378,A -85,B 0,C 180,E1 -19007.91,E2 -19007.91} C_VEL
LIN {X 0,Y 282.985,Z 487.02,A -85,B 0,C 180,E1 -19010.773,E2 -19010.773} C_VEL
LIN {X 0,Y 273.939,Z 476.018,A -85,B 0,C 180,E1 -19013.215,E2 -19013.215} C_VEL
LIN {X 0,Y 266.991,Z 465.493,A -85,B 0,C 180,E1 -19015.198,E2 -19015.198} C_VEL
LIN {X 0,Y 262.19,Z 456.216,A -85,B 0,C 180,E1 -19016.659,E2 -19016.659} C_VEL
LIN {X 0,Y 257.157,Z 444.054,A -85,B 0,C 180,E1 -19018.192,E2 -19018.192} C_VEL
LIN {X 0,Y 252.293,Z 433.786,A -85,B 0,C 180,E1 -19019.373,E2 -19019.373} C_VEL
LIN {X 0,Y 249.275,Z 428.086,A -85,B 0,C 180,E1 -19019.989,E2 -19019.989} C_VEL
LIN {X 0,Y 249.038,Z 426.985,A -85,B 0,C 180,E1 -19020.057,E2 -19020.057} C_VEL
LIN {X 0,Y 249.056,Z 426.961,A -85,B 0,C 180,E1 -19024.358,E2 -19024.358} C_VEL
LIN {X 0,Y 249.033,Z 426.964,A -85,B 0,C 180,E1 -19028.378,E2 -19028.378} C_VEL
LIN {X 0,Y 249.006,Z 426.967,A -85,B 0,C 180,E1 -19032.793,E2 -19032.793} C_VEL
LIN {X 0,Y 249.012,Z 426.967,A -85,B 0,C 180,E1 -19037.363,E2 -19037.363} C_VEL
LIN {X 0,Y 249.037,Z 426.962,A -85,B 0,C 180,E1 -19042.201,E2 -19042.201} C_VEL
LIN {X 0,Y 249.037,Z 426.963,A -85,B 0,C 180,E1 -19045.64,E2 -19045.64} C_VEL
LIN {X 0,Y 249.046,Z 426.963,A -85,B 0,C 180,E1 -19049.473,E2 -19049.473} C_VEL
LIN {X 0,Y 249.068,Z 426.96,A -85,B 0,C 180,E1 -19053.163,E2 -19053.163} C_VEL
LIN {X 0,Y 249.073,Z 426.958,A -85,B 0,C 180,E1 -19056.733,E2 -19056.733} C_VEL
LIN {X 0,Y 249.104,Z 426.95,A -85,B 0,C 180,E1 -19060.212,E2 -19060.212} C_VEL
LIN {X 0,Y 249.237,Z 426.937,A -85,B 0,C 180,E1 -19063.623,E2 -19063.623} C_VEL
LIN {X 0,Y 249.238,Z 426.94,A -85,B 0,C 180,E1 -19068.617,E2 -19068.617} C_VEL
LIN {X 0,Y 249.449,Z 426.91,A -85,B 0,C 180,E1 -19071.903,E2 -19071.903} C_VEL
LIN {X 0,Y 249.291,Z 426.926,A -85,B 0,C 180,E1 -19075.149,E2 -19075.149} C_VEL
LIN {X 0,Y 249.67,Z 426.864,A -85,B 0,C 180,E1 -19078.388,E2 -19078.388} C_VEL
LIN {X 0,Y 249.671,Z 426.88,A -85,B 0,C 180,E1 -19081.614,E2 -19081.614} C_VEL
LIN {X 0,Y 249.449,Z 426.914,A -85,B 0,C 180,E1 -19086.472,E2 -19086.472} C_VEL
LIN {X 0,Y 249.339,Z 426.926,A -85,B 0,C 180,E1 -19089.737,E2 -19089.737} C_VEL
LIN {X 0,Y 249.193,Z 426.946,A -85,B 0,C 180,E1 -19094.705,E2 -19094.705} C_VEL
LIN {X 0,Y 249.131,Z 426.954,A -85,B 0,C 180,E1 -19098.079,E2 -19098.079} C_VEL
LIN {X 0,Y 249.081,Z 426.958,A -85,B 0,C 180,E1 -19101.52,E2 -19101.52} C_VEL
LIN {X 0,Y 249.115,Z 426.956,A -85,B 0,C 180,E1 -19105.477,E2 -19105.477} C_VEL
LIN {X 0,Y 249.082,Z 426.96,A -85,B 0,C 180,E1 -19108.995,E2 -19108.995} C_VEL
LIN {X 0,Y 249.085,Z 427.243,A -85,B 0,C 180,E1 -19110.523,E2 -19110.523} C_VEL
LIN {X 0,Y 249.381,Z 429.495,A -85,B 0,C 180,E1 -19115.189,E2 -19115.189} C_VEL
LIN {X 0,Y 249.62,Z 431.134,A -85,B 0,C 180,E1 -19118.274,E2 -19118.274} C_VEL
LIN {X 0,Y 249.991,Z 433.559,A -85,B 0,C 180,E1 -19122.433,E2 -19122.433} C_VEL
LIN {X 0,Y 250.068,Z 435.852,A -85,B 0,C 180,E1 -19125.996,E2 -19125.996} C_VEL
LIN {X 0,Y 249.853,Z 438.432,A -85,B 0,C 180,E1 -19129.689,E2 -19129.689} C_VEL
LIN {X 0,Y 249.333,Z 440.804,A -85,B 0,C 180,E1 -19132.867,E2 -19132.867} C_VEL
LIN {X 0,Y 248.501,Z 441.551,A -85,B 0,C 180,E1 -19133.743,E2 -19133.743} C_VEL
LIN {X 0,Y 245.417,Z 442.878,A -85,B 0,C 180,E1 -19135.096,E2 -19135.096} C_VEL
LIN {X 0,Y 242.34,Z 444.216,A -85,B 0,C 180,E1 -19136.48,E2 -19136.48} C_VEL
LIN {X 0,Y 241.556,Z 444.98,A -85,B 0,C 180,E1 -19137.393,E2 -19137.393} C_VEL
LIN {X 0,Y 241.251,Z 446.411,A -85,B 0,C 180,E1 -19139.192,E2 -19139.192} C_VEL
LIN {X 0,Y 242.09,Z 449.563,A -85,B 0,C 180,E1 -19139.456,E2 -19139.456} C_VEL
LIN {X 0,Y 246.104,Z 463.24,A -85,B 0,C 180,E1 -19140.957,E2 -19140.957} C_VEL
LIN {X 0,Y 248.219,Z 473.03,A -85,B 0,C 180,E1 -19142.155,E2 -19142.155} C_VEL
LIN {X 0,Y 249.813,Z 483.264,A -85,B 0,C 180,E1 -19143.566,E2 -19143.566} C_VEL
LIN {X 0,Y 250.504,Z 492.223,A -85,B 0,C 180,E1 -19144.938,E2 -19144.938} C_VEL
LIN {X 0,Y 250.64,Z 500.942,A -85,B 0,C 180,E1 -19146.449,E2 -19146.449} C_VEL
LIN {X 0,Y 248.724,Z 509.469,A -85,B 0,C 180,E1 -19148.014,E2 -19148.014} C_VEL
LIN {X 0,Y 246.998,Z 516.686,A -85,B 0,C 180,E1 -19149.601,E2 -19149.601} C_VEL
LIN {X 0,Y 245.739,Z 522.618,A -85,B 0,C 180,E1 -19151.146,E2 -19151.146} C_VEL
LIN {X 0,Y 243.967,Z 529.428,A -85,B 0,C 180,E1 -19153.258,E2 -19153.258} C_VEL
LIN {X 0,Y 242.835,Z 533.929,A -85,B 0,C 180,E1 -19154.902,E2 -19154.902} C_VEL
LIN {X 0,Y 241.493,Z 539.421,A -85,B 0,C 180,E1 -19157.393,E2 -19157.393} C_VEL
LIN {X 0,Y 240.64,Z 543.751,A -85,B 0,C 180,E1 -19159.908,E2 -19159.908} C_VEL
LIN {X 0,Y 240.223,Z 546.121,A -85,B 0,C 180,E1 -19161.589,E2 -19161.589} C_VEL
LIN {X 0,Y 239.955,Z 547.923,A -85,B 0,C 180,E1 -19163.272,E2 -19163.272} C_VEL
LIN {X 0,Y 239.77,Z 550.376,A -85,B 0,C 180,E1 -19166.639,E2 -19166.639} C_VEL
LIN {X 0,Y 239.818,Z 550.969,A -85,B 0,C 180,E1 -19168.321,E2 -19168.321} C_VEL
LIN {X 0,Y 239.891,Z 551.126,A -85,B 0,C 180,E1 -19170,E2 -19170} C_VEL
LIN {X 0,Y 239.819,Z 550.969,A -85,B 0,C 180,E1 -19171.679,E2 -19171.679} C_VEL
LIN {X 0,Y 239.771,Z 550.376,A -85,B 0,C 180,E1 -19173.361,E2 -19173.361} C_VEL
LIN {X 0,Y 239.955,Z 547.923,A -85,B 0,C 180,E1 -19176.728,E2 -19176.728} C_VEL
LIN {X 0,Y 240.418,Z 544.97,A -85,B 0,C 180,E1 -19179.252,E2 -19179.252} C_VEL
LIN {X 0,Y 241.182,Z 540.977,A -85,B 0,C 180,E1 -19181.769,E2 -19181.769} C_VEL
LIN {X 0,Y 242.323,Z 535.844,A -85,B 0,C 180,E1 -19184.271,E2 -19184.271} C_VEL
LIN {X 0,Y 243.698,Z 530.584,A -85,B 0,C 180,E1 -19186.33,E2 -19186.33} C_VEL
LIN {X 0,Y 245.285,Z 524.268,A -85,B 0,C 180,E1 -19188.371,E2 -19188.371} C_VEL
LIN {X 0,Y 246.594,Z 518.312,A -85,B 0,C 180,E1 -19189.998,E2 -19189.998} C_VEL
LIN {X 0,Y 248.199,Z 511.386,A -85,B 0,C 180,E1 -19191.598,E2 -19191.598} C_VEL
LIN {X 0,Y 250.135,Z 503.211,A -85,B 0,C 180,E1 -19193.163,E2 -19193.163} C_VEL
LIN {X 0,Y 250.751,Z 499.803,A -85,B 0,C 180,E1 -19193.759,E2 -19193.759} C_VEL
LIN {X 0,Y 250.254,Z 487.961,A -85,B 0,C 180,E1 -19195.744,E2 -19195.744} C_VEL
LIN {X 0,Y 249.198,Z 478.634,A -85,B 0,C 180,E1 -19197.099,E2 -19197.099} C_VEL
LIN {X 0,Y 247.057,Z 467.267,A -85,B 0,C 180,E1 -19198.561,E2 -19198.561} C_VEL
LIN {X 0,Y 244.224,Z 456.35,A -85,B 0,C 180,E1 -19199.812,E2 -19199.812} C_VEL
LIN {X 0,Y 241.333,Z 447.1,A -85,B 0,C 180,E1 -19200.761,E2 -19200.761} C_VEL
LIN {X 0,Y 241.267,Z 446.409,A -85,B 0,C 180,E1 -19200.84,E2 -19200.84} C_VEL
LIN {X 0,Y 242.038,Z 442.754,A -85,B 0,C 180,E1 -19205.501,E2 -19205.501} C_VEL
LIN {X 0,Y 242.646,Z 439.75,A -85,B 0,C 180,E1 -19209.583,E2 -19209.583} C_VEL
LIN {X 0,Y 243.033,Z 436.915,A -85,B 0,C 180,E1 -19213.701,E2 -19213.701} C_VEL
LIN {X 0,Y 243.002,Z 435.265,A -85,B 0,C 180,E1 -19216.305,E2 -19216.305} C_VEL
LIN {X 0,Y 242.666,Z 432.863,A -85,B 0,C 180,E1 -19220.419,E2 -19220.419} C_VEL
LIN {X 0,Y 242.368,Z 430.668,A -85,B 0,C 180,E1 -19224.552,E2 -19224.552} C_VEL
LIN {X 0,Y 242.126,Z 428.778,A -85,B 0,C 180,E1 -19228.501,E2 -19228.501} C_VEL
LIN {X 0,Y 242.039,Z 427.866,A -85,B 0,C 180,E1 -19230.584,E2 -19230.584} C_VEL
LIN {X 0,Y 242.066,Z 427.834,A -85,B 0,C 180,E1 -19234.182,E2 -19234.182} C_VEL
LIN {X 0,Y 242.023,Z 427.839,A -85,B 0,C 180,E1 -19238.312,E2 -19238.312} C_VEL
LIN {X 0,Y 242.16,Z 427.821,A -85,B 0,C 180,E1 -19243.277,E2 -19243.277} C_VEL
LIN {X 0,Y 242.176,Z 427.818,A -85,B 0,C 180,E1 -19248.278,E2 -19248.278} C_VEL
LIN {X 0,Y 242.396,Z 427.792,A -85,B 0,C 180,E1 -19251.664,E2 -19251.664} C_VEL
LIN {X 0,Y 242.253,Z 427.808,A -85,B 0,C 180,E1 -19255.006,E2 -19255.006} C_VEL
LIN {X 0,Y 242.631,Z 427.757,A -85,B 0,C 180,E1 -19258.339,E2 -19258.339} C_VEL
LIN {X 0,Y 242.631,Z 427.74,A -85,B 0,C 180,E1 -19261.659,E2 -19261.659} C_VEL
LIN {X 0,Y 242.416,Z 427.787,A -85,B 0,C 180,E1 -19266.681,E2 -19266.681} C_VEL
LIN {X 0,Y 242.262,Z 427.804,A -85,B 0,C 180,E1 -19270.023,E2 -19270.023} C_VEL
LIN {X 0,Y 242.158,Z 427.817,A -85,B 0,C 180,E1 -19275.14,E2 -19275.14} C_VEL
LIN {X 0,Y 242.067,Z 427.831,A -85,B 0,C 180,E1 -19278.624,E2 -19278.624} C_VEL
LIN {X 0,Y 242.007,Z 427.838,A -85,B 0,C 180,E1 -19282.179,E2 -19282.179} C_VEL
LIN {X 0,Y 242.061,Z 427.83,A -85,B 0,C 180,E1 -19285.838,E2 -19285.838} C_VEL
LIN {X 0,Y 242.025,Z 427.837,A -85,B 0,C 180,E1 -19289.58,E2 -19289.58} C_VEL
LIN {X 0,Y 241.985,Z 427.841,A -85,B 0,C 180,E1 -19293.491,E2 -19293.491} C_VEL
LIN {X 0,Y 242.007,Z 427.838,A -85,B 0,C 180,E1 -19297.577,E2 -19297.577} C_VEL
LIN {X 0,Y 241.993,Z 427.84,A -85,B 0,C 180,E1 -19301.909,E2 -19301.909} C_VEL
LIN {X 0,Y 241.937,Z 427.847,A -85,B 0,C 180,E1 -19305.801,E2 -19305.801} C_VEL
LIN {X 0,Y 241.968,Z 427.844,A -85,B 0,C 180,E1 -19310.284,E2 -19310.284} C_VEL
LIN {X 0,Y 242.032,Z 427.838,A -85,B 0,C 180,E1 -19314.498,E2 -19314.498} C_VEL
LIN {X 0,Y 242.026,Z 428.015,A -85,B 0,C 180,E1 -19319.005,E2 -19319.005} C_VEL
LIN {X 0,Y 243.116,Z 430.887,A -85,B 0,C 180,E1 -19319.279,E2 -19319.279} C_VEL
LIN {X 0,Y 248.832,Z 441.89,A -85,B 0,C 180,E1 -19320.616,E2 -19320.616} C_VEL
LIN {X 0,Y 253.479,Z 452.844,A -85,B 0,C 180,E1 -19322.024,E2 -19322.024} C_VEL
LIN {X 0,Y 256.345,Z 459.974,A -85,B 0,C 180,E1 -19323.034,E2 -19323.034} C_VEL
LIN {X 0,Y 261.118,Z 469.37,A -85,B 0,C 180,E1 -19324.636,E2 -19324.636} C_VEL
LIN {X 0,Y 267.785,Z 479.608,A -85,B 0,C 180,E1 -19326.716,E2 -19326.716} C_VEL
LIN {X 0,Y 276.033,Z 489.774,A -85,B 0,C 180,E1 -19329.118,E2 -19329.118} C_VEL
LIN {X 0,Y 285.088,Z 499.173,A -85,B 0,C 180,E1 -19331.636,E2 -19331.636} C_VEL
LIN {X 0,Y 293.975,Z 507.59,A -85,B 0,C 180,E1 -19334.136,E2 -19334.136} C_VEL
LIN {X 0,Y 300.002,Z 512.943,A -85,B 0,C 180,E1 -19335.888,E2 -19335.888} C_VEL
LIN {X 0,Y 306.899,Z 519.112,A -85,B 0,C 180,E1 -19338.106,E2 -19338.106} C_VEL
LIN {X 0,Y 312.531,Z 523.975,A -85,B 0,C 180,E1 -19340.198,E2 -19340.198} C_VEL
LIN {X 0,Y 315.992,Z 526.847,A -85,B 0,C 180,E1 -19341.688,E2 -19341.688} C_VEL
LIN {X 0,Y 319.332,Z 529.79,A -85,B 0,C 180,E1 -19343.682,E2 -19343.682} C_VEL
LIN {X 0,Y 321.227,Z 531.281,A -85,B 0,C 180,E1 -19344.979,E2 -19344.979} C_VEL
LIN {X 0,Y 323.75,Z 532.76,A -85,B 0,C 180,E1 -19346.922,E2 -19346.922} C_VEL
LIN {X 0,Y 325.488,Z 533.325,A -85,B 0,C 180,E1 -19348.763,E2 -19348.763} C_VEL
LIN {X 0,Y 325.953,Z 533.404,A -85,B 0,C 180,E1 -19350,E2 -19350} C_VEL
LIN {X 0,Y 325.456,Z 533.333,A -85,B 0,C 180,E1 -19351.237,E2 -19351.237} C_VEL
LIN {X 0,Y 323.751,Z 532.756,A -85,B 0,C 180,E1 -19353.079,E2 -19353.079} C_VEL
LIN {X 0,Y 321.232,Z 531.274,A -85,B 0,C 180,E1 -19355.02,E2 -19355.02} C_VEL
LIN {X 0,Y 318.52,Z 529.123,A -85,B 0,C 180,E1 -19356.837,E2 -19356.837} C_VEL
LIN {X 0,Y 315.982,Z 526.854,A -85,B 0,C 180,E1 -19358.312,E2 -19358.312} C_VEL
LIN {X 0,Y 312.474,Z 523.98,A -85,B 0,C 180,E1 -19359.792,E2 -19359.792} C_VEL
LIN {X 0,Y 308.278,Z 520.363,A -85,B 0,C 180,E1 -19361.397,E2 -19361.397} C_VEL
LIN {X 0,Y 302.032,Z 514.849,A -85,B 0,C 180,E1 -19363.455,E2 -19363.455} C_VEL
LIN {X 0,Y 295.2,Z 508.718,A -85,B 0,C 180,E1 -19365.504,E2 -19365.504} C_VEL
LIN {X 0,Y 286.357,Z 500.443,A -85,B 0,C 180,E1 -19368.009,E2 -19368.009} C_VEL
LIN {X 0,Y 277.542,Z 491.347,A -85,B 0,C 180,E1 -19370.462,E2 -19370.462} C_VEL
LIN {X 0,Y 268.984,Z 481.182,A -85,B 0,C 180,E1 -19372.93,E2 -19372.93} C_VEL
LIN {X 0,Y 262.423,Z 471.576,A -85,B 0,C 180,E1 -19374.942,E2 -19374.942} C_VEL
LIN {X 0,Y 257.901,Z 463.311,A -85,B 0,C 180,E1 -19376.427,E2 -19376.427} C_VEL
LIN {X 0,Y 254.119,Z 454.525,A -85,B 0,C 180,E1 -19377.75,E2 -19377.75} C_VEL
LIN {X 0,Y 249.415,Z 443.06,A -85,B 0,C 180,E1 -19379.231,E2 -19379.231} C_VEL
LIN {X 0,Y 243.366,Z 431.239,A -85,B 0,C 180,E1 -19380.679,E2 -19380.679} C_VEL
LIN {X 0,Y 242.124,Z 428.549,A -85,B 0,C 180,E1 -19380.963,E2 -19380.963} C_VEL
LIN {X 0,Y 241.987,Z 427.843,A -85,B 0,C 180,E1 -19381.032,E2 -19381.032} C_VEL
LIN {X 0,Y 242.024,Z 427.839,A -85,B 0,C 180,E1 -19385.604,E2 -19385.604} C_VEL
LIN {X 0,Y 241.967,Z 427.845,A -85,B 0,C 180,E1 -19389.716,E2 -19389.716} C_VEL
LIN {X 0,Y 241.928,Z 427.848,A -85,B 0,C 180,E1 -19394.201,E2 -19394.201} C_VEL
LIN {X 0,Y 241.933,Z 427.848,A -85,B 0,C 180,E1 -19398.078,E2 -19398.078} C_VEL
LIN {X 0,Y 241.98,Z 427.841,A -85,B 0,C 180,E1 -19402.418,E2 -19402.418} C_VEL
LIN {X 0,Y 241.975,Z 427.843,A -85,B 0,C 180,E1 -19406.508,E2 -19406.508} C_VEL
LIN {X 0,Y 242.031,Z 427.837,A -85,B 0,C 180,E1 -19410.588,E2 -19410.588} C_VEL
LIN {X 0,Y 242.062,Z 427.83,A -85,B 0,C 180,E1 -19414.183,E2 -19414.183} C_VEL
LIN {X 0,Y 242.048,Z 427.834,A -85,B 0,C 180,E1 -19418.298,E2 -19418.298} C_VEL
LIN {X 0,Y 242.158,Z 427.819,A -85,B 0,C 180,E1 -19423.279,E2 -19423.279} C_VEL
LIN {X 0,Y 242.175,Z 427.819,A -85,B 0,C 180,E1 -19428.28,E2 -19428.28} C_VEL
LIN {X 0,Y 242.395,Z 427.788,A -85,B 0,C 180,E1 -19431.665,E2 -19431.665} C_VEL
LIN {X 0,Y 242.252,Z 427.803,A -85,B 0,C 180,E1 -19435.008,E2 -19435.008} C_VEL
LIN {X 0,Y 242.631,Z 427.74,A -85,B 0,C 180,E1 -19438.341,E2 -19438.341} C_VEL
LIN {X 0,Y 242.631,Z 427.757,A -85,B 0,C 180,E1 -19441.661,E2 -19441.661} C_VEL
LIN {X 0,Y 242.419,Z 427.789,A -85,B 0,C 180,E1 -19446.66,E2 -19446.66} C_VEL
LIN {X 0,Y 242.264,Z 427.809,A -85,B 0,C 180,E1 -19450.025,E2 -19450.025} C_VEL
LIN {X 0,Y 242.153,Z 427.822,A -85,B 0,C 180,E1 -19455.143,E2 -19455.143} C_VEL
LIN {X 0,Y 242.066,Z 427.833,A -85,B 0,C 180,E1 -19458.626,E2 -19458.626} C_VEL
LIN {X 0,Y 242.003,Z 427.842,A -85,B 0,C 180,E1 -19462.182,E2 -19462.182} C_VEL
LIN {X 0,Y 242.065,Z 427.837,A -85,B 0,C 180,E1 -19465.839,E2 -19465.839} C_VEL
LIN {X 0,Y 242.036,Z 427.933,A -85,B 0,C 180,E1 -19469.58,E2 -19469.58} C_VEL
LIN {X 0,Y 242.232,Z 429.691,A -85,B 0,C 180,E1 -19473.454,E2 -19473.454} C_VEL
LIN {X 0,Y 242.511,Z 431.737,A -85,B 0,C 180,E1 -19477.488,E2 -19477.488} C_VEL
LIN {X 0,Y 242.879,Z 434.086,A -85,B 0,C 180,E1 -19481.724,E2 -19481.724} C_VEL
LIN {X 0,Y 243.021,Z 435.428,A -85,B 0,C 180,E1 -19483.954,E2 -19483.954} C_VEL
LIN {X 0,Y 243.031,Z 436.944,A -85,B 0,C 180,E1 -19486.3,E2 -19486.3} C_VEL
LIN {X 0,Y 242.645,Z 439.768,A -85,B 0,C 180,E1 -19490.417,E2 -19490.417} C_VEL
LIN {X 0,Y 242.038,Z 442.757,A -85,B 0,C 180,E1 -19494.499,E2 -19494.499} C_VEL
LIN {X 0,Y 241.556,Z 444.98,A -85,B 0,C 180,E1 -19497.393,E2 -19497.393} C_VEL
LIN {X 0,Y 241.481,Z 446.469,A -85,B 0,C 180,E1 -19498.198,E2 -19498.198} C_VEL
LIN {X 0,Y 241.416,Z 449.057,A -85,B 0,C 180,E1 -19498.85,E2 -19498.85} C_VEL
LIN {X 0,Y 241.285,Z 454.102,A -85,B 0,C 180,E1 -19499.576,E2 -19499.576} C_VEL
LIN {X 0,Y 241.138,Z 470.304,A -85,B 0,C 180,E1 -19500.975,E2 -19500.975} C_VEL
LIN {X 0,Y 241.324,Z 472.208,A -85,B 0,C 180,E1 -19501.216,E2 -19501.216} C_VEL
LIN {X 0,Y 242.891,Z 482.194,A -85,B 0,C 180,E1 -19502.63,E2 -19502.63} C_VEL
LIN {X 0,Y 243.794,Z 492.051,A -85,B 0,C 180,E1 -19504.204,E2 -19504.204} C_VEL
LIN {X 0,Y 243.988,Z 500.74,A -85,B 0,C 180,E1 -19505.766,E2 -19505.766} C_VEL
LIN {X 0,Y 242.119,Z 509.271,A -85,B 0,C 180,E1 -19507.381,E2 -19507.381} C_VEL
LIN {X 0,Y 240.334,Z 516.488,A -85,B 0,C 180,E1 -19509.009,E2 -19509.009} C_VEL
LIN {X 0,Y 238.915,Z 522.729,A -85,B 0,C 180,E1 -19510.686,E2 -19510.686} C_VEL
LIN {X 0,Y 237.134,Z 529.229,A -85,B 0,C 180,E1 -19512.761,E2 -19512.761} C_VEL
LIN {X 0,Y 235.957,Z 533.731,A -85,B 0,C 180,E1 -19514.451,E2 -19514.451} C_VEL
LIN {X 0,Y 234.537,Z 539.224,A -85,B 0,C 180,E1 -19517.013,E2 -19517.013} C_VEL
LIN {X 0,Y 233.611,Z 543.553,A -85,B 0,C 180,E1 -19519.601,E2 -19519.601} C_VEL
LIN {X 0,Y 233.193,Z 545.923,A -85,B 0,C 180,E1 -19521.333,E2 -19521.333} C_VEL
LIN {X 0,Y 232.893,Z 547.725,A -85,B 0,C 180,E1 -19523.067,E2 -19523.067} C_VEL
LIN {X 0,Y 232.679,Z 550.179,A -85,B 0,C 180,E1 -19526.537,E2 -19526.537} C_VEL
LIN {X 0,Y 232.732,Z 550.772,A -85,B 0,C 180,E1 -19528.27,E2 -19528.27} C_VEL
LIN {X 0,Y 232.802,Z 550.93,A -85,B 0,C 180,E1 -19530,E2 -19530} C_VEL
LIN {X 0,Y 232.732,Z 550.772,A -85,B 0,C 180,E1 -19531.73,E2 -19531.73} C_VEL
LIN {X 0,Y 232.692,Z 549.494,A -85,B 0,C 180,E1 -19534.647,E2 -19534.647} C_VEL
LIN {X 0,Y 232.893,Z 547.725,A -85,B 0,C 180,E1 -19536.933,E2 -19536.933} C_VEL
LIN {X 0,Y 233.396,Z 544.772,A -85,B 0,C 180,E1 -19539.533,E2 -19539.533} C_VEL
LIN {X 0,Y 234.194,Z 540.779,A -85,B 0,C 180,E1 -19542.126,E2 -19542.126} C_VEL
LIN {X 0,Y 235.422,Z 535.647,A -85,B 0,C 180,E1 -19544.699,E2 -19544.699} C_VEL
LIN {X 0,Y 236.87,Z 530.386,A -85,B 0,C 180,E1 -19546.815,E2 -19546.815} C_VEL
LIN {X 0,Y 238.542,Z 524.07,A -85,B 0,C 180,E1 -19548.91,E2 -19548.91} C_VEL
LIN {X 0,Y 239.892,Z 518.114,A -85,B 0,C 180,E1 -19550.582,E2 -19550.582} C_VEL
LIN {X 0,Y 241.603,Z 511.189,A -85,B 0,C 180,E1 -19552.219,E2 -19552.219} C_VEL
LIN {X 0,Y 243.609,Z 503.013,A -85,B 0,C 180,E1 -19553.821,E2 -19553.821} C_VEL
LIN {X 0,Y 244.021,Z 498.448,A -85,B 0,C 180,E1 -19554.683,E2 -19554.683} C_VEL
LIN {X 0,Y 243.518,Z 487.603,A -85,B 0,C 180,E1 -19556.532,E2 -19556.532} C_VEL
LIN {X 0,Y 242.358,Z 478.354,A -85,B 0,C 180,E1 -19557.938,E2 -19557.938} C_VEL
LIN {X 0,Y 240.619,Z 468.732,A -85,B 0,C 180,E1 -19559.244,E2 -19559.244} C_VEL
LIN {X 0,Y 237.53,Z 456.815,A -85,B 0,C 180,E1 -19560.694,E2 -19560.694} C_VEL
LIN {X 0,Y 234.524,Z 447.35,A -85,B 0,C 180,E1 -19561.734,E2 -19561.734} C_VEL
LIN {X 0,Y 234.384,Z 446.211,A -85,B 0,C 180,E1 -19561.871,E2 -19561.871} C_VEL
LIN {X 0,Y 235.125,Z 442.563,A -85,B 0,C 180,E1 -19566.712,E2 -19566.712} C_VEL
LIN {X 0,Y 235.514,Z 440.863,A -85,B 0,C 180,E1 -19569.115,E2 -19569.115} C_VEL
LIN {X 0,Y 235.93,Z 438.078,A -85,B 0,C 180,E1 -19573.245,E2 -19573.245} C_VEL
LIN {X 0,Y 235.928,Z 435.912,A -85,B 0,C 180,E1 -19576.752,E2 -19576.752} C_VEL
LIN {X 0,Y 235.619,Z 433.605,A -85,B 0,C 180,E1 -19580.851,E2 -19580.851} C_VEL
LIN {X 0,Y 235.262,Z 431.294,A -85,B 0,C 180,E1 -19585.417,E2 -19585.417} C_VEL
LIN {X 0,Y 235.042,Z 429.17,A -85,B 0,C 180,E1 -19590.125,E2 -19590.125} C_VEL
LIN {X 0,Y 234.949,Z 428.721,A -85,B 0,C 180,E1 -19591.405,E2 -19591.405} C_VEL
LIN {X 0,Y 234.975,Z 428.717,A -85,B 0,C 180,E1 -19595.244,E2 -19595.244} C_VEL
LIN {X 0,Y 234.995,Z 428.714,A -85,B 0,C 180,E1 -19598.967,E2 -19598.967} C_VEL
LIN {X 0,Y 235.093,Z 428.701,A -85,B 0,C 180,E1 -19603.059,E2 -19603.059} C_VEL
LIN {X 0,Y 235.109,Z 428.7,A -85,B 0,C 180,E1 -19607.921,E2 -19607.921} C_VEL
LIN {X 0,Y 235.327,Z 428.673,A -85,B 0,C 180,E1 -19611.411,E2 -19611.411} C_VEL
LIN {X 0,Y 235.369,Z 428.665,A -85,B 0,C 180,E1 -19613.139,E2 -19613.139} C_VEL
LIN {X 0,Y 235.591,Z 428.634,A -85,B 0,C 180,E1 -19618.29,E2 -19618.29} C_VEL
LIN {X 0,Y 235.591,Z 428.615,A -85,B 0,C 180,E1 -19621.709,E2 -19621.709} C_VEL
LIN {X 0,Y 235.387,Z 428.664,A -85,B 0,C 180,E1 -19626.858,E2 -19626.858} C_VEL
LIN {X 0,Y 235.209,Z 428.682,A -85,B 0,C 180,E1 -19630.327,E2 -19630.327} C_VEL
LIN {X 0,Y 235.106,Z 428.697,A -85,B 0,C 180,E1 -19635.606,E2 -19635.606} C_VEL
LIN {X 0,Y 235.003,Z 428.708,A -85,B 0,C 180,E1 -19639.205,E2 -19639.205} C_VEL
LIN {X 0,Y 234.956,Z 428.719,A -85,B 0,C 180,E1 -19642.882,E2 -19642.882} C_VEL
LIN {X 0,Y 234.964,Z 428.715,A -85,B 0,C 180,E1 -19646.657,E2 -19646.657} C_VEL
LIN {X 0,Y 234.927,Z 428.722,A -85,B 0,C 180,E1 -19650.567,E2 -19650.567} C_VEL
LIN {X 0,Y 234.955,Z 428.719,A -85,B 0,C 180,E1 -19654.633,E2 -19654.633} C_VEL
LIN {X 0,Y 234.961,Z 428.719,A -85,B 0,C 180,E1 -19658.952,E2 -19658.952} C_VEL
LIN {X 0,Y 234.969,Z 428.716,A -85,B 0,C 180,E1 -19663.466,E2 -19663.466} C_VEL
LIN {X 0,Y 234.917,Z 428.724,A -85,B 0,C 180,E1 -19668.409,E2 -19668.409} C_VEL
LIN {X 0,Y 234.95,Z 428.72,A -85,B 0,C 180,E1 -19671.086,E2 -19671.086} C_VEL
LIN {X 0,Y 234.956,Z 428.718,A -85,B 0,C 180,E1 -19675.367,E2 -19675.367} C_VEL
LIN {X 0,Y 234.933,Z 428.727,A -85,B 0,C 180,E1 -19677.977,E2 -19677.977} C_VEL
LIN {X 0,Y 235.85,Z 431.445,A -85,B 0,C 180,E1 -19678.239,E2 -19678.239} C_VEL
LIN {X 0,Y 237.136,Z 433.637,A -85,B 0,C 180,E1 -19678.536,E2 -19678.536} C_VEL
LIN {X 0,Y 242.421,Z 443.883,A -85,B 0,C 180,E1 -19679.882,E2 -19679.882} C_VEL
LIN {X 0,Y 246.463,Z 453.325,A -85,B 0,C 180,E1 -19681.178,E2 -19681.178} C_VEL
LIN {X 0,Y 249.819,Z 462.324,A -85,B 0,C 180,E1 -19682.509,E2 -19682.509} C_VEL
LIN {X 0,Y 253.99,Z 471.021,A -85,B 0,C 180,E1 -19684.061,E2 -19684.061} C_VEL
LIN {X 0,Y 259.759,Z 480.506,A -85,B 0,C 180,E1 -19686.057,E2 -19686.057} C_VEL
LIN {X 0,Y 267.891,Z 490.985,A -85,B 0,C 180,E1 -19688.638,E2 -19688.638} C_VEL
LIN {X 0,Y 276.518,Z 500.224,A -85,B 0,C 180,E1 -19691.215,E2 -19691.215} C_VEL
LIN {X 0,Y 285.412,Z 508.446,A -85,B 0,C 180,E1 -19693.806,E2 -19693.806} C_VEL
LIN {X 0,Y 293.201,Z 515.1,A -85,B 0,C 180,E1 -19696.132,E2 -19696.132} C_VEL
LIN {X 0,Y 299.969,Z 520.767,A -85,B 0,C 180,E1 -19698.344,E2 -19698.344} C_VEL
LIN {X 0,Y 306.241,Z 525.926,A -85,B 0,C 180,E1 -19700.681,E2 -19700.681} C_VEL
LIN {X 0,Y 309.618,Z 528.685,A -85,B 0,C 180,E1 -19702.173,E2 -19702.173} C_VEL
LIN {X 0,Y 311.89,Z 530.737,A -85,B 0,C 180,E1 -19703.531,E2 -19703.531} C_VEL
LIN {X 0,Y 313.89,Z 532.386,A -85,B 0,C 180,E1 -19704.862,E2 -19704.862} C_VEL
LIN {X 0,Y 316.701,Z 534.117,A -85,B 0,C 180,E1 -19706.96,E2 -19706.96} C_VEL
LIN {X 0,Y 318.435,Z 534.704,A -85,B 0,C 180,E1 -19708.735,E2 -19708.735} C_VEL
LIN {X 0,Y 318.983,Z 534.817,A -85,B 0,C 180,E1 -19710,E2 -19710} C_VEL
LIN {X 0,Y 318.412,Z 534.709,A -85,B 0,C 180,E1 -19711.265,E2 -19711.265} C_VEL
LIN {X 0,Y 316.701,Z 534.112,A -85,B 0,C 180,E1 -19713.041,E2 -19713.041} C_VEL
LIN {X 0,Y 313.89,Z 532.376,A -85,B 0,C 180,E1 -19715.138,E2 -19715.138} C_VEL
LIN {X 0,Y 311.404,Z 530.306,A -85,B 0,C 180,E1 -19716.779,E2 -19716.779} C_VEL
LIN {X 0,Y 309.591,Z 528.686,A -85,B 0,C 180,E1 -19717.828,E2 -19717.828} C_VEL
LIN {X 0,Y 306.219,Z 525.986,A -85,B 0,C 180,E1 -19719.293,E2 -19719.293} C_VEL
LIN {X 0,Y 300.996,Z 521.649,A -85,B 0,C 180,E1 -19721.29,E2 -19721.29} C_VEL
LIN {X 0,Y 294.941,Z 516.623,A -85,B 0,C 180,E1 -19723.31,E2 -19723.31} C_VEL
LIN {X 0,Y 287.378,Z 510.219,A -85,B 0,C 180,E1 -19725.605,E2 -19725.605} C_VEL
LIN {X 0,Y 277.771,Z 501.436,A -85,B 0,C 180,E1 -19728.416,E2 -19728.416} C_VEL
LIN {X 0,Y 269.107,Z 492.329,A -85,B 0,C 180,E1 -19730.993,E2 -19730.993} C_VEL
LIN {X 0,Y 261.622,Z 483.193,A -85,B 0,C 180,E1 -19733.319,E2 -19733.319} C_VEL
LIN {X 0,Y 256.213,Z 474.957,A -85,B 0,C 180,E1 -19735.152,E2 -19735.152} C_VEL
LIN {X 0,Y 251.831,Z 466.713,A -85,B 0,C 180,E1 -19736.744,E2 -19736.744} C_VEL
LIN {X 0,Y 247.636,Z 456.426,A -85,B 0,C 180,E1 -19738.385,E2 -19738.385} C_VEL
LIN {X 0,Y 242.994,Z 445.202,A -85,B 0,C 180,E1 -19739.948,E2 -19739.948} C_VEL
LIN {X 0,Y 237.588,Z 434.502,A -85,B 0,C 180,E1 -19741.377,E2 -19741.377} C_VEL
LIN {X 0,Y 235.173,Z 429.886,A -85,B 0,C 180,E1 -19741.939,E2 -19741.939} C_VEL
LIN {X 0,Y 234.93,Z 428.722,A -85,B 0,C 180,E1 -19742.073,E2 -19742.073} C_VEL
LIN {X 0,Y 234.951,Z 428.719,A -85,B 0,C 180,E1 -19746.136,E2 -19746.136} C_VEL
LIN {X 0,Y 234.937,Z 428.721,A -85,B 0,C 180,E1 -19748.944,E2 -19748.944} C_VEL
LIN {X 0,Y 234.884,Z 428.728,A -85,B 0,C 180,E1 -19753.485,E2 -19753.485} C_VEL
LIN {X 0,Y 234.884,Z 428.726,A -85,B 0,C 180,E1 -19756.515,E2 -19756.515} C_VEL
LIN {X 0,Y 234.912,Z 428.725,A -85,B 0,C 180,E1 -19761.079,E2 -19761.079} C_VEL
LIN {X 0,Y 234.921,Z 428.723,A -85,B 0,C 180,E1 -19765.362,E2 -19765.362} C_VEL
LIN {X 0,Y 234.926,Z 428.722,A -85,B 0,C 180,E1 -19769.433,E2 -19769.433} C_VEL
LIN {X 0,Y 234.989,Z 428.711,A -85,B 0,C 180,E1 -19773.794,E2 -19773.794} C_VEL
LIN {X 0,Y 235.006,Z 428.709,A -85,B 0,C 180,E1 -19778.97,E2 -19778.97} C_VEL
LIN {X 0,Y 235.091,Z 428.701,A -85,B 0,C 180,E1 -19783.06,E2 -19783.06} C_VEL
LIN {X 0,Y 235.108,Z 428.698,A -85,B 0,C 180,E1 -19787.923,E2 -19787.923} C_VEL
LIN {X 0,Y 235.326,Z 428.669,A -85,B 0,C 180,E1 -19791.413,E2 -19791.413} C_VEL
LIN {X 0,Y 235.368,Z 428.666,A -85,B 0,C 180,E1 -19793.141,E2 -19793.141} C_VEL
LIN {X 0,Y 235.591,Z 428.615,A -85,B 0,C 180,E1 -19798.291,E2 -19798.291} C_VEL
LIN {X 0,Y 235.591,Z 428.634,A -85,B 0,C 180,E1 -19801.71,E2 -19801.71} C_VEL
LIN {X 0,Y 235.369,Z 428.667,A -85,B 0,C 180,E1 -19806.861,E2 -19806.861} C_VEL
LIN {X 0,Y 235.21,Z 428.689,A -85,B 0,C 180,E1 -19810.329,E2 -19810.329} C_VEL
LIN {X 0,Y 235.104,Z 428.7,A -85,B 0,C 180,E1 -19815.608,E2 -19815.608} C_VEL
LIN {X 0,Y 235.002,Z 428.712,A -85,B 0,C 180,E1 -19819.207,E2 -19819.207} C_VEL
LIN {X 0,Y 234.95,Z 428.721,A -85,B 0,C 180,E1 -19822.885,E2 -19822.885} C_VEL
LIN {X 0,Y 234.967,Z 428.719,A -85,B 0,C 180,E1 -19826.659,E2 -19826.659} C_VEL
LIN {X 0,Y 234.949,Z 428.72,A -85,B 0,C 180,E1 -19828.595,E2 -19828.595} C_VEL
LIN {X 0,Y 235.162,Z 430.338,A -85,B 0,C 180,E1 -19832.545,E2 -19832.545} C_VEL
LIN {X 0,Y 235.418,Z 432.32,A -85,B 0,C 180,E1 -19836.661,E2 -19836.661} C_VEL
LIN {X 0,Y 235.795,Z 434.621,A -85,B 0,C 180,E1 -19840.976,E2 -19840.976} C_VEL
LIN {X 0,Y 235.968,Z 436.598,A -85,B 0,C 180,E1 -19844.374,E2 -19844.374} C_VEL
LIN {X 0,Y 235.842,Z 439.02,A -85,B 0,C 180,E1 -19848.159,E2 -19848.159} C_VEL
LIN {X 0,Y 235.491,Z 441.089,A -85,B 0,C 180,E1 -19851.192,E2 -19851.192} C_VEL
LIN {X 0,Y 234.792,Z 444.085,A -85,B 0,C 180,E1 -19855.34,E2 -19855.34} C_VEL
LIN {X 0,Y 234.366,Z 446.224,A -85,B 0,C 180,E1 -19858.18,E2 -19858.18} C_VEL
LIN {X 0,Y 235.209,Z 449.401,A -85,B 0,C 180,E1 -19858.465,E2 -19858.465} C_VEL
LIN {X 0,Y 238.865,Z 461.467,A -85,B 0,C 180,E1 -19859.844,E2 -19859.844} C_VEL
LIN {X 0,Y 241.324,Z 472.208,A -85,B 0,C 180,E1 -19861.216,E2 -19861.216} C_VEL
LIN {X 0,Y 241.518,Z 477.694,A -85,B 0,C 180,E1 -19861.873,E2 -19861.873} C_VEL
LIN {X 0,Y 239.9,Z 486.38,A -85,B 0,C 180,E1 -19862.876,E2 -19862.876} C_VEL
LIN {X 0,Y 237.81,Z 494.897,A -85,B 0,C 180,E1 -19864.005,E2 -19864.005} C_VEL
LIN {X 0,Y 237.277,Z 499.65,A -85,B 0,C 180,E1 -19864.854,E2 -19864.854} C_VEL
LIN {X 0,Y 237.116,Z 502.816,A -85,B 0,C 180,E1 -19865.484,E2 -19865.484} C_VEL
LIN {X 0,Y 235.096,Z 510.993,A -85,B 0,C 180,E1 -19867.132,E2 -19867.132} C_VEL
LIN {X 0,Y 232.73,Z 519.958,A -85,B 0,C 180,E1 -19869.335,E2 -19869.335} C_VEL
LIN {X 0,Y 230.651,Z 527.875,A -85,B 0,C 180,E1 -19871.801,E2 -19871.801} C_VEL
LIN {X 0,Y 229.1,Z 533.533,A -85,B 0,C 180,E1 -19873.973,E2 -19873.973} C_VEL
LIN {X 0,Y 227.574,Z 539.025,A -85,B 0,C 180,E1 -19876.608,E2 -19876.608} C_VEL
LIN {X 0,Y 226.604,Z 543.355,A -85,B 0,C 180,E1 -19879.276,E2 -19879.276} C_VEL
LIN {X 0,Y 226.152,Z 545.726,A -85,B 0,C 180,E1 -19881.061,E2 -19881.061} C_VEL
LIN {X 0,Y 225.825,Z 547.528,A -85,B 0,C 180,E1 -19882.849,E2 -19882.849} C_VEL
LIN {X 0,Y 225.593,Z 549.982,A -85,B 0,C 180,E1 -19886.428,E2 -19886.428} C_VEL
LIN {X 0,Y 225.628,Z 550.575,A -85,B 0,C 180,E1 -19888.215,E2 -19888.215} C_VEL
LIN {X 0,Y 225.714,Z 550.733,A -85,B 0,C 180,E1 -19890,E2 -19890} C_VEL
LIN {X 0,Y 225.628,Z 550.575,A -85,B 0,C 180,E1 -19891.785,E2 -19891.785} C_VEL
LIN {X 0,Y 225.592,Z 549.498,A -85,B 0,C 180,E1 -19894.49,E2 -19894.49} C_VEL
LIN {X 0,Y 225.825,Z 547.528,A -85,B 0,C 180,E1 -19897.151,E2 -19897.151} C_VEL
LIN {X 0,Y 226.358,Z 544.574,A -85,B 0,C 180,E1 -19899.832,E2 -19899.832} C_VEL
LIN {X 0,Y 227.226,Z 540.581,A -85,B 0,C 180,E1 -19902.504,E2 -19902.504} C_VEL
LIN {X 0,Y 228.539,Z 535.449,A -85,B 0,C 180,E1 -19905.152,E2 -19905.152} C_VEL
LIN {X 0,Y 230.036,Z 530.188,A -85,B 0,C 180,E1 -19907.33,E2 -19907.33} C_VEL
LIN {X 0,Y 231.796,Z 523.872,A -85,B 0,C 180,E1 -19909.482,E2 -19909.482} C_VEL
LIN {X 0,Y 233.226,Z 517.916,A -85,B 0,C 180,E1 -19911.198,E2 -19911.198} C_VEL
LIN {X 0,Y 235.03,Z 510.991,A -85,B 0,C 180,E1 -19912.875,E2 -19912.875} C_VEL
LIN {X 0,Y 237.105,Z 502.815,A -85,B 0,C 180,E1 -19914.517,E2 -19914.517} C_VEL
LIN {X 0,Y 237.209,Z 495.611,A -85,B 0,C 180,E1 -19915.913,E2 -19915.913} C_VEL
LIN {X 0,Y 236.724,Z 486.563,A -85,B 0,C 180,E1 -19917.477,E2 -19917.477} C_VEL
LIN {X 0,Y 235.275,Z 476.094,A -85,B 0,C 180,E1 -19919.102,E2 -19919.102} C_VEL
LIN {X 0,Y 233.553,Z 467.353,A -85,B 0,C 180,E1 -19920.33,E2 -19920.33} C_VEL
LIN {X 0,Y 230.598,Z 456.208,A -85,B 0,C 180,E1 -19921.75,E2 -19921.75} C_VEL
LIN {X 0,Y 227.591,Z 447.098,A -85,B 0,C 180,E1 -19922.821,E2 -19922.821} C_VEL
LIN {X 0,Y 227.457,Z 446.055,A -85,B 0,C 180,E1 -19922.923,E2 -19922.923} C_VEL
LIN {X 0,Y 228.059,Z 443.254,A -85,B 0,C 180,E1 -19926.751,E2 -19926.751} C_VEL
LIN {X 0,Y 228.555,Z 440.899,A -85,B 0,C 180,E1 -19930.22,E2 -19930.22} C_VEL
LIN {X 0,Y 228.815,Z 439.4,A -85,B 0,C 180,E1 -19932.509,E2 -19932.509} C_VEL
LIN {X 0,Y 228.912,Z 437.819,A -85,B 0,C 180,E1 -19935.077,E2 -19935.077} C_VEL
LIN {X 0,Y 228.844,Z 436.398,A -85,B 0,C 180,E1 -19937.495,E2 -19937.495} C_VEL
LIN {X 0,Y 228.449,Z 433.99,A -85,B 0,C 180,E1 -19942.027,E2 -19942.027} C_VEL
LIN {X 0,Y 228.204,Z 431.917,A -85,B 0,C 180,E1 -19946.333,E2 -19946.333} C_VEL
LIN {X 0,Y 227.991,Z 430.141,A -85,B 0,C 180,E1 -19950.447,E2 -19950.447} C_VEL
LIN {X 0,Y 227.941,Z 429.593,A -85,B 0,C 180,E1 -19953.396,E2 -19953.396} C_VEL
LIN {X 0,Y 227.945,Z 429.593,A -85,B 0,C 180,E1 -19958.284,E2 -19958.284} C_VEL
LIN {X 0,Y 228.031,Z 429.58,A -85,B 0,C 180,E1 -19962.825,E2 -19962.825} C_VEL
LIN {X 0,Y 228.067,Z 429.578,A -85,B 0,C 180,E1 -19967.542,E2 -19967.542} C_VEL
LIN {X 0,Y 228.263,Z 429.551,A -85,B 0,C 180,E1 -19971.143,E2 -19971.143} C_VEL
LIN {X 0,Y 228.32,Z 429.542,A -85,B 0,C 180,E1 -19972.927,E2 -19972.927} C_VEL
LIN {X 0,Y 228.55,Z 429.511,A -85,B 0,C 180,E1 -19978.237,E2 -19978.237} C_VEL
LIN {X 0,Y 228.549,Z 429.491,A -85,B 0,C 180,E1 -19981.761,E2 -19981.761} C_VEL
LIN {X 0,Y 228.334,Z 429.543,A -85,B 0,C 180,E1 -19987.071,E2 -19987.071} C_VEL
LIN {X 0,Y 228.14,Z 429.563,A -85,B 0,C 180,E1 -19990.65,E2 -19990.65} C_VEL
LIN {X 0,Y 228.057,Z 429.572,A -85,B 0,C 180,E1 -19994.272,E2 -19994.272} C_VEL
LIN {X 0,Y 227.998,Z 429.583,A -85,B 0,C 180,E1 -19997.953,E2 -19997.953} C_VEL
LIN {X 0,Y 227.925,Z 429.593,A -85,B 0,C 180,E1 -20002.328,E2 -20002.328} C_VEL
LIN {X 0,Y 227.938,Z 429.59,A -85,B 0,C 180,E1 -20006.602,E2 -20006.602} C_VEL
LIN {X 0,Y 227.903,Z 429.596,A -85,B 0,C 180,E1 -20010.296,E2 -20010.296} C_VEL
LIN {X 0,Y 227.884,Z 429.597,A -85,B 0,C 180,E1 -20013.718,E2 -20013.718} C_VEL
LIN {X 0,Y 227.866,Z 429.599,A -85,B 0,C 180,E1 -20018.085,E2 -20018.085} C_VEL
LIN {X 0,Y 227.911,Z 429.595,A -85,B 0,C 180,E1 -20022.718,E2 -20022.718} C_VEL
LIN {X 0,Y 227.843,Z 429.603,A -85,B 0,C 180,E1 -20027.755,E2 -20027.755} C_VEL
LIN {X 0,Y 227.865,Z 429.601,A -85,B 0,C 180,E1 -20031.914,E2 -20031.914} C_VEL
LIN {X 0,Y 227.886,Z 429.6,A -85,B 0,C 180,E1 -20036.373,E2 -20036.373} C_VEL
LIN {X 0,Y 227.918,Z 429.703,A -85,B 0,C 180,E1 -20036.898,E2 -20036.898} C_VEL
LIN {X 0,Y 228.975,Z 432.554,A -85,B 0,C 180,E1 -20037.211,E2 -20037.211} C_VEL
LIN {X 0,Y 233.725,Z 441.33,A -85,B 0,C 180,E1 -20038.434,E2 -20038.434} C_VEL
LIN {X 0,Y 238.526,Z 451.647,A -85,B 0,C 180,E1 -20039.942,E2 -20039.942} C_VEL
LIN {X 0,Y 242.642,Z 462.632,A -85,B 0,C 180,E1 -20041.635,E2 -20041.635} C_VEL
LIN {X 0,Y 246.681,Z 472.165,A -85,B 0,C 180,E1 -20043.363,E2 -20043.363} C_VEL
LIN {X 0,Y 251.431,Z 480.75,A -85,B 0,C 180,E1 -20045.211,E2 -20045.211} C_VEL
LIN {X 0,Y 256.972,Z 488.72,A -85,B 0,C 180,E1 -20047.183,E2 -20047.183} C_VEL
LIN {X 0,Y 265.03,Z 498.163,A -85,B 0,C 180,E1 -20049.835,E2 -20049.835} C_VEL
LIN {X 0,Y 274.848,Z 507.588,A -85,B 0,C 180,E1 -20052.85,E2 -20052.85} C_VEL
LIN {X 0,Y 283.207,Z 514.711,A -85,B 0,C 180,E1 -20055.42,E2 -20055.42} C_VEL
LIN {X 0,Y 289.376,Z 519.611,A -85,B 0,C 180,E1 -20057.375,E2 -20057.375} C_VEL
LIN {X 0,Y 294.091,Z 523.223,A -85,B 0,C 180,E1 -20058.979,E2 -20058.979} C_VEL
LIN {X 0,Y 298.985,Z 526.981,A -85,B 0,C 180,E1 -20060.838,E2 -20060.838} C_VEL
LIN {X 0,Y 301.731,Z 528.964,A -85,B 0,C 180,E1 -20061.967,E2 -20061.967} C_VEL
LIN {X 0,Y 304.323,Z 531.132,A -85,B 0,C 180,E1 -20063.369,E2 -20063.369} C_VEL
LIN {X 0,Y 306.398,Z 532.871,A -85,B 0,C 180,E1 -20064.736,E2 -20064.736} C_VEL
LIN {X 0,Y 308.301,Z 534.186,A -85,B 0,C 180,E1 -20066.079,E2 -20066.079} C_VEL
LIN {X 0,Y 309.992,Z 535.047,A -85,B 0,C 180,E1 -20067.401,E2 -20067.401} C_VEL
LIN {X 0,Y 311.265,Z 535.533,A -85,B 0,C 180,E1 -20068.706,E2 -20068.706} C_VEL
LIN {X 0,Y 311.909,Z 535.689,A -85,B 0,C 180,E1 -20070,E2 -20070} C_VEL
LIN {X 0,Y 311.248,Z 535.535,A -85,B 0,C 180,E1 -20071.294,E2 -20071.294} C_VEL
LIN {X 0,Y 309.628,Z 534.866,A -85,B 0,C 180,E1 -20072.916,E2 -20072.916} C_VEL
LIN {X 0,Y 308.303,Z 534.185,A -85,B 0,C 180,E1 -20073.921,E2 -20073.921} C_VEL
LIN {X 0,Y 306.398,Z 532.871,A -85,B 0,C 180,E1 -20075.264,E2 -20075.264} C_VEL
LIN {X 0,Y 303.1,Z 530.083,A -85,B 0,C 180,E1 -20077.326,E2 -20077.326} C_VEL
LIN {X 0,Y 301.686,Z 528.966,A -85,B 0,C 180,E1 -20078.035,E2 -20078.035} C_VEL
LIN {X 0,Y 296.159,Z 524.859,A -85,B 0,C 180,E1 -20080.252,E2 -20080.252} C_VEL
LIN {X 0,Y 291.835,Z 521.468,A -85,B 0,C 180,E1 -20081.811,E2 -20081.811} C_VEL
LIN {X 0,Y 285.827,Z 516.755,A -85,B 0,C 180,E1 -20083.782,E2 -20083.782} C_VEL
LIN {X 0,Y 278.045,Z 510.421,A -85,B 0,C 180,E1 -20086.16,E2 -20086.16} C_VEL
LIN {X 0,Y 269.945,Z 503.109,A -85,B 0,C 180,E1 -20088.63,E2 -20088.63} C_VEL
LIN {X 0,Y 261.903,Z 494.67,A -85,B 0,C 180,E1 -20091.176,E2 -20091.176} C_VEL
LIN {X 0,Y 254.656,Z 485.637,A -85,B 0,C 180,E1 -20093.606,E2 -20093.606} C_VEL
LIN {X 0,Y 248.609,Z 475.841,A -85,B 0,C 180,E1 -20095.884,E2 -20095.884} C_VEL
LIN {X 0,Y 244.354,Z 466.903,A -85,B 0,C 180,E1 -20097.636,E2 -20097.636} C_VEL
LIN {X 0,Y 239.877,Z 454.945,A -85,B 0,C 180,E1 -20099.557,E2 -20099.557} C_VEL
LIN {X 0,Y 235.525,Z 445.072,A -85,B 0,C 180,E1 -20101.025,E2 -20101.025} C_VEL
LIN {X 0,Y 230.82,Z 435.84,A -85,B 0,C 180,E1 -20102.349,E2 -20102.349} C_VEL
LIN {X 0,Y 228.072,Z 430.499,A -85,B 0,C 180,E1 -20103.042,E2 -20103.042} C_VEL
LIN {X 0,Y 227.899,Z 429.598,A -85,B 0,C 180,E1 -20103.155,E2 -20103.155} C_VEL
LIN {X 0,Y 227.9,Z 429.597,A -85,B 0,C 180,E1 -20106.7,E2 -20106.7} C_VEL
LIN {X 0,Y 227.829,Z 429.604,A -85,B 0,C 180,E1 -20110.375,E2 -20110.375} C_VEL
LIN {X 0,Y 227.83,Z 429.605,A -85,B 0,C 180,E1 -20115.192,E2 -20115.192} C_VEL
LIN {X 0,Y 227.821,Z 429.606,A -85,B 0,C 180,E1 -20119.624,E2 -20119.624} C_VEL
LIN {X 0,Y 227.874,Z 429.598,A -85,B 0,C 180,E1 -20124.128,E2 -20124.128} C_VEL
LIN {X 0,Y 227.865,Z 429.601,A -85,B 0,C 180,E1 -20128.378,E2 -20128.378} C_VEL
LIN {X 0,Y 227.881,Z 429.599,A -85,B 0,C 180,E1 -20132.446,E2 -20132.446} C_VEL
LIN {X 0,Y 227.909,Z 429.592,A -85,B 0,C 180,E1 -20136.368,E2 -20136.368} C_VEL
LIN {X 0,Y 227.937,Z 429.586,A -85,B 0,C 180,E1 -20140.175,E2 -20140.175} C_VEL
LIN {X 0,Y 228.051,Z 429.576,A -85,B 0,C 180,E1 -20143.898,E2 -20143.898} C_VEL
LIN {X 0,Y 228.066,Z 429.575,A -85,B 0,C 180,E1 -20147.544,E2 -20147.544} C_VEL
LIN {X 0,Y 228.262,Z 429.549,A -85,B 0,C 180,E1 -20151.145,E2 -20151.145} C_VEL
LIN {X 0,Y 228.319,Z 429.545,A -85,B 0,C 180,E1 -20152.928,E2 -20152.928} C_VEL
LIN {X 0,Y 228.549,Z 429.491,A -85,B 0,C 180,E1 -20158.239,E2 -20158.239} C_VEL
LIN {X 0,Y 228.55,Z 429.511,A -85,B 0,C 180,E1 -20161.763,E2 -20161.763} C_VEL
LIN {X 0,Y 228.32,Z 429.544,A -85,B 0,C 180,E1 -20167.073,E2 -20167.073} C_VEL
LIN {X 0,Y 228.142,Z 429.568,A -85,B 0,C 180,E1 -20170.652,E2 -20170.652} C_VEL
LIN {X 0,Y 228.056,Z 429.581,A -85,B 0,C 180,E1 -20174.274,E2 -20174.274} C_VEL
LIN {X 0,Y 227.999,Z 429.587,A -85,B 0,C 180,E1 -20177.955,E2 -20177.955} C_VEL
LIN {X 0,Y 227.914,Z 429.598,A -85,B 0,C 180,E1 -20182.322,E2 -20182.322} C_VEL
LIN {X 0,Y 227.941,Z 429.595,A -85,B 0,C 180,E1 -20186.604,E2 -20186.604} C_VEL
LIN {X 0,Y 227.991,Z 430.137,A -85,B 0,C 180,E1 -20189.553,E2 -20189.553} C_VEL
LIN {X 0,Y 228.199,Z 431.954,A -85,B 0,C 180,E1 -20193.745,E2 -20193.745} C_VEL
LIN {X 0,Y 228.451,Z 434.002,A -85,B 0,C 180,E1 -20197.973,E2 -20197.973} C_VEL
LIN {X 0,Y 228.671,Z 435.15,A -85,B 0,C 180,E1 -20200.198,E2 -20200.198} C_VEL
LIN {X 0,Y 228.842,Z 436.432,A -85,B 0,C 180,E1 -20202.519,E2 -20202.519} C_VEL
LIN {X 0,Y 228.915,Z 437.923,A -85,B 0,C 180,E1 -20205.08,E2 -20205.08} C_VEL
LIN {X 0,Y 228.815,Z 439.414,A -85,B 0,C 180,E1 -20207.491,E2 -20207.491} C_VEL
LIN {X 0,Y 228.268,Z 442.424,A -85,B 0,C 180,E1 -20211.993,E2 -20211.993} C_VEL
LIN {X 0,Y 227.487,Z 445.967,A -85,B 0,C 180,E1 -20217.006,E2 -20217.006} C_VEL
LIN {X 0,Y 227.513,Z 446.517,A -85,B 0,C 180,E1 -20217.138,E2 -20217.138} C_VEL
LIN {X 0,Y 228.534,Z 449.67,A -85,B 0,C 180,E1 -20217.46,E2 -20217.46} C_VEL
LIN {X 0,Y 232.401,Z 462.801,A -85,B 0,C 180,E1 -20219.064,E2 -20219.064} C_VEL
LIN {X 0,Y 234.797,Z 473.268,A -85,B 0,C 180,E1 -20220.491,E2 -20220.491} C_VEL
LIN {X 0,Y 236.34,Z 483.526,A -85,B 0,C 180,E1 -20222.031,E2 -20222.031} C_VEL
LIN {X 0,Y 237.093,Z 491.927,A -85,B 0,C 180,E1 -20223.433,E2 -20223.433} C_VEL
LIN {X 0,Y 237.277,Z 499.65,A -85,B 0,C 180,E1 -20224.854,E2 -20224.854} C_VEL
LIN {X 0,Y 236.802,Z 502.799,A -85,B 0,C 180,E1 -20225.439,E2 -20225.439} C_VEL
LIN {X 0,Y 234.774,Z 507.401,A -85,B 0,C 180,E1 -20226.222,E2 -20226.222} C_VEL
LIN {X 0,Y 227.112,Z 518.399,A -85,B 0,C 180,E1 -20228.369,E2 -20228.369} C_VEL
LIN {X 0,Y 225.634,Z 521.621,A -85,B 0,C 180,E1 -20229.252,E2 -20229.252} C_VEL
LIN {X 0,Y 225.478,Z 522.221,A -85,B 0,C 180,E1 -20229.447,E2 -20229.447} C_VEL
LIN {X 0,Y 223.525,Z 528.833,A -85,B 0,C 180,E1 -20231.675,E2 -20231.675} C_VEL
LIN {X 0,Y 222.269,Z 533.336,A -85,B 0,C 180,E1 -20233.467,E2 -20233.467} C_VEL
LIN {X 0,Y 220.636,Z 538.827,A -85,B 0,C 180,E1 -20236.179,E2 -20236.179} C_VEL
LIN {X 0,Y 219.612,Z 543.158,A -85,B 0,C 180,E1 -20238.93,E2 -20238.93} C_VEL
LIN {X 0,Y 219.104,Z 545.528,A -85,B 0,C 180,E1 -20240.771,E2 -20240.771} C_VEL
LIN {X 0,Y 218.764,Z 547.33,A -85,B 0,C 180,E1 -20242.617,E2 -20242.617} C_VEL
LIN {X 0,Y 218.501,Z 549.785,A -85,B 0,C 180,E1 -20246.312,E2 -20246.312} C_VEL
LIN {X 0,Y 218.527,Z 550.378,A -85,B 0,C 180,E1 -20248.157,E2 -20248.157} C_VEL
LIN {X 0,Y 218.629,Z 550.536,A -85,B 0,C 180,E1 -20250,E2 -20250} C_VEL
LIN {X 0,Y 218.527,Z 550.378,A -85,B 0,C 180,E1 -20251.843,E2 -20251.843} C_VEL
LIN {X 0,Y 218.489,Z 549.511,A -85,B 0,C 180,E1 -20254.308,E2 -20254.308} C_VEL
LIN {X 0,Y 218.764,Z 547.33,A -85,B 0,C 180,E1 -20257.383,E2 -20257.383} C_VEL
LIN {X 0,Y 219.341,Z 544.376,A -85,B 0,C 180,E1 -20260.15,E2 -20260.15} C_VEL
LIN {X 0,Y 220.246,Z 540.383,A -85,B 0,C 180,E1 -20262.907,E2 -20262.907} C_VEL
LIN {X 0,Y 221.677,Z 535.251,A -85,B 0,C 180,E1 -20265.633,E2 -20265.633} C_VEL
LIN {X 0,Y 223.225,Z 529.99,A -85,B 0,C 180,E1 -20267.876,E2 -20267.876} C_VEL
LIN {X 0,Y 225.068,Z 523.674,A -85,B 0,C 180,E1 -20270.089,E2 -20270.089} C_VEL
LIN {X 0,Y 226.58,Z 517.718,A -85,B 0,C 180,E1 -20271.852,E2 -20271.852} C_VEL
LIN {X 0,Y 228.483,Z 510.794,A -85,B 0,C 180,E1 -20273.57,E2 -20273.57} C_VEL
LIN {X 0,Y 230.379,Z 503.752,A -85,B 0,C 180,E1 -20275.041,E2 -20275.041} C_VEL
LIN {X 0,Y 230.514,Z 495.404,A -85,B 0,C 180,E1 -20276.724,E2 -20276.724} C_VEL
LIN {X 0,Y 230.072,Z 486.905,A -85,B 0,C 180,E1 -20278.259,E2 -20278.259} C_VEL
LIN {X 0,Y 228.815,Z 477.484,A -85,B 0,C 180,E1 -20279.807,E2 -20279.807} C_VEL
LIN {X 0,Y 227.003,Z 468.056,A -85,B 0,C 180,E1 -20281.21,E2 -20281.21} C_VEL
LIN {X 0,Y 223.811,Z 456.14,A -85,B 0,C 180,E1 -20282.819,E2 -20282.819} C_VEL
LIN {X 0,Y 221.396,Z 449.026,A -85,B 0,C 180,E1 -20283.751,E2 -20283.751} C_VEL
LIN {X 0,Y 220.56,Z 445.858,A -85,B 0,C 180,E1 -20284.107,E2 -20284.107} C_VEL
LIN {X 0,Y 221.067,Z 443.554,A -85,B 0,C 180,E1 -20287.364,E2 -20287.364} C_VEL
LIN {X 0,Y 221.633,Z 440.722,A -85,B 0,C 180,E1 -20291.751,E2 -20291.751} C_VEL
LIN {X 0,Y 221.817,Z 439.228,A -85,B 0,C 180,E1 -20294.189,E2 -20294.189} C_VEL
LIN {X 0,Y 221.714,Z 436.906,A -85,B 0,C 180,E1 -20298.265,E2 -20298.265} C_VEL
LIN {X 0,Y 221.369,Z 434.561,A -85,B 0,C 180,E1 -20302.899,E2 -20302.899} C_VEL
LIN {X 0,Y 221.09,Z 432.55,A -85,B 0,C 180,E1 -20307.288,E2 -20307.288} C_VEL
LIN {X 0,Y 221.039,Z 431.656,A -85,B 0,C 180,E1 -20309.42,E2 -20309.42} C_VEL
LIN {X 0,Y 220.884,Z 430.472,A -85,B 0,C 180,E1 -20312.983,E2 -20312.983} C_VEL
LIN {X 0,Y 220.863,Z 430.476,A -85,B 0,C 180,E1 -20317.551,E2 -20317.551} C_VEL
LIN {X 0,Y 220.981,Z 430.458,A -85,B 0,C 180,E1 -20322.571,E2 -20322.571} C_VEL
LIN {X 0,Y 221.006,Z 430.456,A -85,B 0,C 180,E1 -20327.137,E2 -20327.137} C_VEL
LIN {X 0,Y 221.201,Z 430.43,A -85,B 0,C 180,E1 -20330.858,E2 -20330.858} C_VEL
LIN {X 0,Y 221.255,Z 430.422,A -85,B 0,C 180,E1 -20332.699,E2 -20332.699} C_VEL
LIN {X 0,Y 221.508,Z 430.388,A -85,B 0,C 180,E1 -20338.181,E2 -20338.181} C_VEL
LIN {X 0,Y 221.507,Z 430.366,A -85,B 0,C 180,E1 -20341.817,E2 -20341.817} C_VEL
LIN {X 0,Y 221.267,Z 430.425,A -85,B 0,C 180,E1 -20347.298,E2 -20347.298} C_VEL
LIN {X 0,Y 221.062,Z 430.446,A -85,B 0,C 180,E1 -20350.996,E2 -20350.996} C_VEL
LIN {X 0,Y 221.011,Z 430.453,A -85,B 0,C 180,E1 -20356.629,E2 -20356.629} C_VEL
LIN {X 0,Y 220.887,Z 430.464,A -85,B 0,C 180,E1 -20360.485,E2 -20360.485} C_VEL
LIN {X 0,Y 220.862,Z 430.469,A -85,B 0,C 180,E1 -20364.434,E2 -20364.434} C_VEL
LIN {X 0,Y 220.831,Z 430.477,A -85,B 0,C 180,E1 -20368.513,E2 -20368.513} C_VEL
LIN {X 0,Y 220.819,Z 430.48,A -85,B 0,C 180,E1 -20372.754,E2 -20372.754} C_VEL
LIN {X 0,Y 220.833,Z 430.477,A -85,B 0,C 180,E1 -20377.288,E2 -20377.288} C_VEL
LIN {X 0,Y 220.855,Z 430.474,A -85,B 0,C 180,E1 -20381.931,E2 -20381.931} C_VEL
LIN {X 0,Y 220.787,Z 430.482,A -85,B 0,C 180,E1 -20385.551,E2 -20385.551} C_VEL
LIN {X 0,Y 220.797,Z 430.48,A -85,B 0,C 180,E1 -20389.81,E2 -20389.81} C_VEL
LIN {X 0,Y 220.827,Z 430.479,A -85,B 0,C 180,E1 -20392.794,E2 -20392.794} C_VEL
LIN {X 0,Y 220.85,Z 430.602,A -85,B 0,C 180,E1 -20395.727,E2 -20395.727} C_VEL
LIN {X 0,Y 221.94,Z 433.501,A -85,B 0,C 180,E1 -20396.07,E2 -20396.07} C_VEL
LIN {X 0,Y 223.345,Z 435.82,A -85,B 0,C 180,E1 -20396.431,E2 -20396.431} C_VEL
LIN {X 0,Y 228.246,Z 445.162,A -85,B 0,C 180,E1 -20397.859,E2 -20397.859} C_VEL
LIN {X 0,Y 232.658,Z 455.009,A -85,B 0,C 180,E1 -20399.415,E2 -20399.415} C_VEL
LIN {X 0,Y 236.105,Z 464.45,A -85,B 0,C 180,E1 -20400.973,E2 -20400.973} C_VEL
LIN {X 0,Y 239.063,Z 472.253,A -85,B 0,C 180,E1 -20402.423,E2 -20402.423} C_VEL
LIN {X 0,Y 243.963,Z 482.091,A -85,B 0,C 180,E1 -20404.59,E2 -20404.59} C_VEL
LIN {X 0,Y 250.179,Z 491.471,A -85,B 0,C 180,E1 -20407.03,E2 -20407.03} C_VEL
LIN {X 0,Y 258.242,Z 500.907,A -85,B 0,C 180,E1 -20409.864,E2 -20409.864} C_VEL
LIN {X 0,Y 267.413,Z 509.519,A -85,B 0,C 180,E1 -20412.838,E2 -20412.838} C_VEL
LIN {X 0,Y 275.847,Z 516.396,A -85,B 0,C 180,E1 -20415.499,E2 -20415.499} C_VEL
LIN {X 0,Y 283.255,Z 521.941,A -85,B 0,C 180,E1 -20417.915,E2 -20417.915} C_VEL
LIN {X 0,Y 289.71,Z 526.556,A -85,B 0,C 180,E1 -20420.223,E2 -20420.223} C_VEL
LIN {X 0,Y 295.29,Z 530.3,A -85,B 0,C 180,E1 -20422.478,E2 -20422.478} C_VEL
LIN {X 0,Y 297.101,Z 531.695,A -85,B 0,C 180,E1 -20423.465,E2 -20423.465} C_VEL
LIN {X 0,Y 300.85,Z 534.411,A -85,B 0,C 180,E1 -20425.981,E2 -20425.981} C_VEL
LIN {X 0,Y 302.683,Z 535.352,A -85,B 0,C 180,E1 -20427.338,E2 -20427.338} C_VEL
LIN {X 0,Y 304.049,Z 535.911,A -85,B 0,C 180,E1 -20428.676,E2 -20428.676} C_VEL
LIN {X 0,Y 304.806,Z 536.095,A -85,B 0,C 180,E1 -20430,E2 -20430} C_VEL
LIN {X 0,Y 304.038,Z 535.912,A -85,B 0,C 180,E1 -20431.325,E2 -20431.325} C_VEL
LIN {X 0,Y 302.55,Z 535.292,A -85,B 0,C 180,E1 -20432.761,E2 -20432.761} C_VEL
LIN {X 0,Y 300.852,Z 534.411,A -85,B 0,C 180,E1 -20434.019,E2 -20434.019} C_VEL
LIN {X 0,Y 297.101,Z 531.697,A -85,B 0,C 180,E1 -20436.533,E2 -20436.533} C_VEL
LIN {X 0,Y 295.229,Z 530.302,A -85,B 0,C 180,E1 -20437.523,E2 -20437.523} C_VEL
LIN {X 0,Y 289.702,Z 526.556,A -85,B 0,C 180,E1 -20439.777,E2 -20439.777} C_VEL
LIN {X 0,Y 285.411,Z 523.47,A -85,B 0,C 180,E1 -20441.361,E2 -20441.361} C_VEL
LIN {X 0,Y 278.138,Z 518.159,A -85,B 0,C 180,E1 -20443.769,E2 -20443.769} C_VEL
LIN {X 0,Y 270.671,Z 512.332,A -85,B 0,C 180,E1 -20446.118,E2 -20446.118} C_VEL
LIN {X 0,Y 262.494,Z 505.064,A -85,B 0,C 180,E1 -20448.74,E2 -20448.74} C_VEL
LIN {X 0,Y 253.927,Z 496.036,A -85,B 0,C 180,E1 -20451.638,E2 -20451.638} C_VEL
LIN {X 0,Y 248.123,Z 488.576,A -85,B 0,C 180,E1 -20453.759,E2 -20453.759} C_VEL
LIN {X 0,Y 242.497,Z 479.379,A -85,B 0,C 180,E1 -20456.049,E2 -20456.049} C_VEL
LIN {X 0,Y 238.485,Z 470.82,A -85,B 0,C 180,E1 -20457.864,E2 -20457.864} C_VEL
LIN {X 0,Y 234.215,Z 458.931,A -85,B 0,C 180,E1 -20459.955,E2 -20459.955} C_VEL
LIN {X 0,Y 229.122,Z 446.934,A -85,B 0,C 180,E1 -20461.869,E2 -20461.869} C_VEL
LIN {X 0,Y 222.638,Z 434.387,A -85,B 0,C 180,E1 -20463.785,E2 -20463.785} C_VEL
LIN {X 0,Y 221.091,Z 431.716,A -85,B 0,C 180,E1 -20464.181,E2 -20464.181} C_VEL
LIN {X 0,Y 220.819,Z 430.479,A -85,B 0,C 180,E1 -20464.346,E2 -20464.346} C_VEL
LIN {X 0,Y 220.834,Z 430.478,A -85,B 0,C 180,E1 -20467.288,E2 -20467.288} C_VEL
LIN {X 0,Y 220.771,Z 430.484,A -85,B 0,C 180,E1 -20471.951,E2 -20471.951} C_VEL
LIN {X 0,Y 220.77,Z 430.486,A -85,B 0,C 180,E1 -20475.547,E2 -20475.547} C_VEL
LIN {X 0,Y 220.801,Z 430.48,A -85,B 0,C 180,E1 -20480.463,E2 -20480.463} C_VEL
LIN {X 0,Y 220.795,Z 430.483,A -85,B 0,C 180,E1 -20485.045,E2 -20485.045} C_VEL
LIN {X 0,Y 220.863,Z 430.474,A -85,B 0,C 180,E1 -20489.395,E2 -20489.395} C_VEL
LIN {X 0,Y 220.89,Z 430.468,A -85,B 0,C 180,E1 -20493.55,E2 -20493.55} C_VEL
LIN {X 0,Y 220.873,Z 430.472,A -85,B 0,C 180,E1 -20497.554,E2 -20497.554} C_VEL
LIN {X 0,Y 220.979,Z 430.459,A -85,B 0,C 180,E1 -20502.572,E2 -20502.572} C_VEL
LIN {X 0,Y 221.005,Z 430.456,A -85,B 0,C 180,E1 -20507.139,E2 -20507.139} C_VEL
LIN {X 0,Y 221.2,Z 430.427,A -85,B 0,C 180,E1 -20510.86,E2 -20510.86} C_VEL
LIN {X 0,Y 221.254,Z 430.426,A -85,B 0,C 180,E1 -20512.701,E2 -20512.701} C_VEL
LIN {X 0,Y 221.507,Z 430.366,A -85,B 0,C 180,E1 -20518.183,E2 -20518.183} C_VEL
LIN {X 0,Y 221.508,Z 430.388,A -85,B 0,C 180,E1 -20521.819,E2 -20521.819} C_VEL
LIN {X 0,Y 221.255,Z 430.424,A -85,B 0,C 180,E1 -20527.301,E2 -20527.301} C_VEL
LIN {X 0,Y 221.063,Z 430.449,A -85,B 0,C 180,E1 -20530.998,E2 -20530.998} C_VEL
LIN {X 0,Y 221.011,Z 430.457,A -85,B 0,C 180,E1 -20536.631,E2 -20536.631} C_VEL
LIN {X 0,Y 220.881,Z 430.472,A -85,B 0,C 180,E1 -20540.488,E2 -20540.488} C_VEL
LIN {X 0,Y 220.86,Z 430.477,A -85,B 0,C 180,E1 -20544.437,E2 -20544.437} C_VEL
LIN {X 0,Y 220.884,Z 430.473,A -85,B 0,C 180,E1 -20547.017,E2 -20547.017} C_VEL
LIN {X 0,Y 221.029,Z 431.771,A -85,B 0,C 180,E1 -20550.852,E2 -20550.852} C_VEL
LIN {X 0,Y 221.232,Z 433.52,A -85,B 0,C 180,E1 -20554.878,E2 -20554.878} C_VEL
LIN {X 0,Y 221.556,Z 435.702,A -85,B 0,C 180,E1 -20559.378,E2 -20559.378} C_VEL
LIN {X 0,Y 221.781,Z 437.759,A -85,B 0,C 180,E1 -20563.212,E2 -20563.212} C_VEL
LIN {X 0,Y 221.752,Z 439.829,A -85,B 0,C 180,E1 -20566.799,E2 -20566.799} C_VEL
LIN {X 0,Y 221.369,Z 442.226,A -85,B 0,C 180,E1 -20570.584,E2 -20570.584} C_VEL
LIN {X 0,Y 221.066,Z 443.715,A -85,B 0,C 180,E1 -20572.841,E2 -20572.841} C_VEL
LIN {X 0,Y 220.565,Z 445.871,A -85,B 0,C 180,E1 -20575.942,E2 -20575.942} C_VEL
LIN {X 0,Y 221.398,Z 448.996,A -85,B 0,C 180,E1 -20576.248,E2 -20576.248} C_VEL
LIN {X 0,Y 225.295,Z 461.238,A -85,B 0,C 180,E1 -20577.839,E2 -20577.839} C_VEL
LIN {X 0,Y 227.807,Z 471.64,A -85,B 0,C 180,E1 -20579.313,E2 -20579.313} C_VEL
LIN {X 0,Y 229.468,Z 482.118,A -85,B 0,C 180,E1 -20580.934,E2 -20580.934} C_VEL
LIN {X 0,Y 230.417,Z 491.208,A -85,B 0,C 180,E1 -20582.508,E2 -20582.508} C_VEL
LIN {X 0,Y 230.588,Z 500.33,A -85,B 0,C 180,E1 -20584.259,E2 -20584.259} C_VEL
LIN {X 0,Y 230.39,Z 503.753,A -85,B 0,C 180,E1 -20584.96,E2 -20584.96} C_VEL
LIN {X 0,Y 227.547,Z 514.466,A -85,B 0,C 180,E1 -20587.29,E2 -20587.29} C_VEL
LIN {X 0,Y 225.478,Z 522.221,A -85,B 0,C 180,E1 -20589.447,E2 -20589.447} C_VEL
LIN {X 0,Y 223.995,Z 525.91,A -85,B 0,C 180,E1 -20590.583,E2 -20590.583} C_VEL
LIN {X 0,Y 221.503,Z 529.245,A -85,B 0,C 180,E1 -20591.672,E2 -20591.672} C_VEL
LIN {X 0,Y 215.182,Z 536.117,A -85,B 0,C 180,E1 -20594.377,E2 -20594.377} C_VEL
LIN {X 0,Y 213.707,Z 538.674,A -85,B 0,C 180,E1 -20595.749,E2 -20595.749} C_VEL
LIN {X 0,Y 212.615,Z 542.96,A -85,B 0,C 180,E1 -20598.561,E2 -20598.561} C_VEL
LIN {X 0,Y 212.077,Z 545.33,A -85,B 0,C 180,E1 -20600.463,E2 -20600.463} C_VEL
LIN {X 0,Y 211.693,Z 547.132,A -85,B 0,C 180,E1 -20602.369,E2 -20602.369} C_VEL
LIN {X 0,Y 211.42,Z 549.588,A -85,B 0,C 180,E1 -20606.188,E2 -20606.188} C_VEL
LIN {X 0,Y 211.429,Z 550.181,A -85,B 0,C 180,E1 -20608.095,E2 -20608.095} C_VEL
LIN {X 0,Y 211.545,Z 550.34,A -85,B 0,C 180,E1 -20610,E2 -20610} C_VEL
LIN {X 0,Y 211.43,Z 550.181,A -85,B 0,C 180,E1 -20611.905,E2 -20611.905} C_VEL
LIN {X 0,Y 211.396,Z 549.471,A -85,B 0,C 180,E1 -20614.145,E2 -20614.145} C_VEL
LIN {X 0,Y 211.692,Z 547.132,A -85,B 0,C 180,E1 -20617.631,E2 -20617.631} C_VEL
LIN {X 0,Y 212.342,Z 544.179,A -85,B 0,C 180,E1 -20620.488,E2 -20620.488} C_VEL
LIN {X 0,Y 213.282,Z 540.184,A -85,B 0,C 180,E1 -20623.336,E2 -20623.336} C_VEL
LIN {X 0,Y 214.835,Z 535.054,A -85,B 0,C 180,E1 -20626.144,E2 -20626.144} C_VEL
LIN {X 0,Y 216.422,Z 529.791,A -85,B 0,C 180,E1 -20628.458,E2 -20628.458} C_VEL
LIN {X 0,Y 218.376,Z 523.475,A -85,B 0,C 180,E1 -20630.732,E2 -20630.732} C_VEL
LIN {X 0,Y 219.972,Z 517.52,A -85,B 0,C 180,E1 -20632.544,E2 -20632.544} C_VEL
LIN {X 0,Y 221.989,Z 510.596,A -85,B 0,C 180,E1 -20634.303,E2 -20634.303} C_VEL
LIN {X 0,Y 223.865,Z 503.552,A -85,B 0,C 180,E1 -20635.822,E2 -20635.822} C_VEL
LIN {X 0,Y 223.861,Z 495.358,A -85,B 0,C 180,E1 -20637.554,E2 -20637.554} C_VEL
LIN {X 0,Y 223.395,Z 486.78,A -85,B 0,C 180,E1 -20639.17,E2 -20639.17} C_VEL
LIN {X 0,Y 222.054,Z 476.76,A -85,B 0,C 180,E1 -20640.877,E2 -20640.877} C_VEL
LIN {X 0,Y 219.839,Z 466.163,A -85,B 0,C 180,E1 -20642.523,E2 -20642.523} C_VEL
LIN {X 0,Y 217.043,Z 456.054,A -85,B 0,C 180,E1 -20643.968,E2 -20643.968} C_VEL
LIN {X 0,Y 214.48,Z 448.786,A -85,B 0,C 180,E1 -20644.995,E2 -20644.995} C_VEL
LIN {X 0,Y 213.646,Z 445.695,A -85,B 0,C 180,E1 -20645.333,E2 -20645.333} C_VEL
LIN {X 0,Y 214.158,Z 443.507,A -85,B 0,C 180,E1 -20648.573,E2 -20648.573} C_VEL
LIN {X 0,Y 214.497,Z 441.928,A -85,B 0,C 180,E1 -20651.096,E2 -20651.096} C_VEL
LIN {X 0,Y 214.741,Z 440.224,A -85,B 0,C 180,E1 -20653.943,E2 -20653.943} C_VEL
LIN {X 0,Y 214.736,Z 438.741,A -85,B 0,C 180,E1 -20656.582,E2 -20656.582} C_VEL
LIN {X 0,Y 214.625,Z 437.414,A -85,B 0,C 180,E1 -20659.086,E2 -20659.086} C_VEL
LIN {X 0,Y 214.268,Z 435.138,A -85,B 0,C 180,E1 -20663.813,E2 -20663.813} C_VEL
LIN {X 0,Y 214.006,Z 433.055,A -85,B 0,C 180,E1 -20668.63,E2 -20668.63} C_VEL
LIN {X 0,Y 213.843,Z 431.533,A -85,B 0,C 180,E1 -20672.604,E2 -20672.604} C_VEL
LIN {X 0,Y 213.817,Z 431.353,A -85,B 0,C 180,E1 -20676.972,E2 -20676.972} C_VEL
LIN {X 0,Y 213.94,Z 431.336,A -85,B 0,C 180,E1 -20682.802,E2 -20682.802} C_VEL
LIN {X 0,Y 213.947,Z 431.334,A -85,B 0,C 180,E1 -20686.705,E2 -20686.705} C_VEL
LIN {X 0,Y 214.138,Z 431.31,A -85,B 0,C 180,E1 -20690.554,E2 -20690.554} C_VEL
LIN {X 0,Y 214.097,Z 431.315,A -85,B 0,C 180,E1 -20694.347,E2 -20694.347} C_VEL
LIN {X 0,Y 214.441,Z 431.269,A -85,B 0,C 180,E1 -20698.121,E2 -20698.121} C_VEL
LIN {X 0,Y 214.545,Z 431.244,A -85,B 0,C 180,E1 -20699.999,E2 -20699.999} C_VEL
LIN {X 0,Y 214.441,Z 431.245,A -85,B 0,C 180,E1 -20701.877,E2 -20701.877} C_VEL
LIN {X 0,Y 214.203,Z 431.302,A -85,B 0,C 180,E1 -20707.54,E2 -20707.54} C_VEL
LIN {X 0,Y 213.994,Z 431.329,A -85,B 0,C 180,E1 -20711.364,E2 -20711.364} C_VEL
LIN {X 0,Y 213.927,Z 431.332,A -85,B 0,C 180,E1 -20715.236,E2 -20715.236} C_VEL
LIN {X 0,Y 213.927,Z 431.336,A -85,B 0,C 180,E1 -20717.694,E2 -20717.694} C_VEL
LIN {X 0,Y 213.842,Z 431.346,A -85,B 0,C 180,E1 -20723.226,E2 -20723.226} C_VEL
LIN {X 0,Y 213.824,Z 431.35,A -85,B 0,C 180,E1 -20727.449,E2 -20727.449} C_VEL
LIN {X 0,Y 213.774,Z 431.356,A -85,B 0,C 180,E1 -20731.735,E2 -20731.735} C_VEL
LIN {X 0,Y 213.749,Z 431.358,A -85,B 0,C 180,E1 -20736.286,E2 -20736.286} C_VEL
LIN {X 0,Y 213.792,Z 431.355,A -85,B 0,C 180,E1 -20741.105,E2 -20741.105} C_VEL
LIN {X 0,Y 213.804,Z 431.352,A -85,B 0,C 180,E1 -20743.685,E2 -20743.685} C_VEL
LIN {X 0,Y 213.726,Z 431.362,A -85,B 0,C 180,E1 -20748.879,E2 -20748.879} C_VEL
LIN {X 0,Y 213.748,Z 431.36,A -85,B 0,C 180,E1 -20753.713,E2 -20753.713} C_VEL
LIN {X 0,Y 213.763,Z 431.429,A -85,B 0,C 180,E1 -20754.455,E2 -20754.455} C_VEL
LIN {X 0,Y 214.745,Z 434.175,A -85,B 0,C 180,E1 -20754.792,E2 -20754.792} C_VEL
LIN {X 0,Y 216.169,Z 436.353,A -85,B 0,C 180,E1 -20755.176,E2 -20755.176} C_VEL
LIN {X 0,Y 221.035,Z 445.435,A -85,B 0,C 180,E1 -20756.681,E2 -20756.681} C_VEL
LIN {X 0,Y 225.785,Z 455.809,A -85,B 0,C 180,E1 -20758.439,E2 -20758.439} C_VEL
LIN {X 0,Y 229.518,Z 466.02,A -85,B 0,C 180,E1 -20760.231,E2 -20760.231} C_VEL
LIN {X 0,Y 232.588,Z 474.745,A -85,B 0,C 180,E1 -20761.936,E2 -20761.936} C_VEL
LIN {X 0,Y 236.637,Z 483.45,A -85,B 0,C 180,E1 -20763.947,E2 -20763.947} C_VEL
LIN {X 0,Y 241.869,Z 491.961,A -85,B 0,C 180,E1 -20766.243,E2 -20766.243} C_VEL
LIN {X 0,Y 248.629,Z 500.465,A -85,B 0,C 180,E1 -20768.875,E2 -20768.875} C_VEL
LIN {X 0,Y 257.015,Z 508.88,A -85,B 0,C 180,E1 -20771.844,E2 -20771.844} C_VEL
LIN {X 0,Y 266.403,Z 516.561,A -85,B 0,C 180,E1 -20774.938,E2 -20774.938} C_VEL
LIN {X 0,Y 273.724,Z 521.814,A -85,B 0,C 180,E1 -20777.331,E2 -20777.331} C_VEL
LIN {X 0,Y 281.163,Z 526.794,A -85,B 0,C 180,E1 -20779.923,E2 -20779.923} C_VEL
LIN {X 0,Y 287.09,Z 530.529,A -85,B 0,C 180,E1 -20782.262,E2 -20782.262} C_VEL
LIN {X 0,Y 289.942,Z 532.321,A -85,B 0,C 180,E1 -20783.615,E2 -20783.615} C_VEL
LIN {X 0,Y 293.336,Z 534.619,A -85,B 0,C 180,E1 -20785.878,E2 -20785.878} C_VEL
LIN {X 0,Y 295.473,Z 535.639,A -85,B 0,C 180,E1 -20787.409,E2 -20787.409} C_VEL
LIN {X 0,Y 296.776,Z 536.112,A -85,B 0,C 180,E1 -20788.643,E2 -20788.643} C_VEL
LIN {X 0,Y 297.665,Z 536.289,A -85,B 0,C 180,E1 -20790,E2 -20790} C_VEL
LIN {X 0,Y 296.767,Z 536.113,A -85,B 0,C 180,E1 -20791.357,E2 -20791.357} C_VEL
LIN {X 0,Y 295.285,Z 535.558,A -85,B 0,C 180,E1 -20792.728,E2 -20792.728} C_VEL
LIN {X 0,Y 293.337,Z 534.619,A -85,B 0,C 180,E1 -20794.122,E2 -20794.122} C_VEL
LIN {X 0,Y 289.94,Z 532.325,A -85,B 0,C 180,E1 -20796.382,E2 -20796.382} C_VEL
LIN {X 0,Y 287.048,Z 530.53,A -85,B 0,C 180,E1 -20797.739,E2 -20797.739} C_VEL
LIN {X 0,Y 281.174,Z 526.794,A -85,B 0,C 180,E1 -20800.076,E2 -20800.076} C_VEL
LIN {X 0,Y 273.727,Z 521.807,A -85,B 0,C 180,E1 -20802.672,E2 -20802.672} C_VEL
LIN {X 0,Y 265.471,Z 515.891,A -85,B 0,C 180,E1 -20805.351,E2 -20805.351} C_VEL
LIN {X 0,Y 257.015,Z 508.881,A -85,B 0,C 180,E1 -20808.156,E2 -20808.156} C_VEL
LIN {X 0,Y 248.637,Z 500.441,A -85,B 0,C 180,E1 -20811.13,E2 -20811.13} C_VEL
LIN {X 0,Y 241.873,Z 491.95,A -85,B 0,C 180,E1 -20813.759,E2 -20813.759} C_VEL
LIN {X 0,Y 236.652,Z 483.4,A -85,B 0,C 180,E1 -20816.06,E2 -20816.06} C_VEL
LIN {X 0,Y 232.607,Z 474.702,A -85,B 0,C 180,E1 -20818.068,E2 -20818.068} C_VEL
